REGION Network 7: RD 32002
   RUNG wire#powerrail
      { S7_Templates := "SrcType := Int" } EQ_Contact(in1 := "IEC_Counter_0_DB".CV, in2 := 2)
      { S7_Templates := "[card := 0, word_type := UInt, dword_type := UDInt, byte_type := USInt, any_type := Variant]" } "Modbus_Master_DB".Modbus_Master(REQ := wire#w1, MB_ADDR := 1, MODE := 0, DATA_ADDR := 32002, DATA_LEN := 1, DATA_PTR := "Modbus_Send_Receive_1".Reading_Struct."32002", DONE => "Modbus".Done, BUSY => "Modbus".Busy, ERROR => "Modbus".Error, STATUS => "Modbus".Status)
   END_RUNG
   RUNG wire#powerrail
      Contact( "Comm_ok" )
      { S7_Templates := "SrcType := Int" } EQ_Contact(in1 := "IEC_Counter_0_DB".CV, in2 := 2)
      I_Contact( "Modbus_Master_DB".BUSY )
   END_RUNG wire#w1
   // the same network as SCL:
   IF "IEC_Counter_0_DB".CV = 2 THEN
       "Modbus_Master_DB"(REQ := "Comm_ok" AND ("IEC_Counter_0_DB".CV = 2) AND NOT "Modbus_Master_DB".BUSY,   // Modbus_Master
                          MB_ADDR := 1,
                          MODE := 0,
                          DATA_ADDR := 32002,
                          DATA_LEN := 1,
                          DATA_PTR := "Modbus_Send_Receive_1".Reading_Struct."32002",
                          DONE => "Modbus".Done,
                          BUSY => "Modbus".Busy,
                          ERROR => "Modbus".Error,
                          STATUS => "Modbus".Status);
   END_IF;
END_REGION

REGION Network 8: RD 32003
   RUNG wire#powerrail
      { S7_Templates := "SrcType := Int" } EQ_Contact(in1 := "IEC_Counter_0_DB".CV, in2 := 3)
      { S7_Templates := "[card := 0, word_type := UInt, dword_type := UDInt, byte_type := USInt, any_type := Variant]" } "Modbus_Master_DB".Modbus_Master(REQ := wire#w1, MB_ADDR := 1, MODE := 0, DATA_ADDR := 32003, DATA_LEN := 1, DATA_PTR := "Modbus_Send_Receive_1".Reading_Struct."32003", DONE => "Modbus".Done, BUSY => "Modbus".Busy, ERROR => "Modbus".Error, STATUS => "Modbus".Status)
   END_RUNG
   RUNG wire#powerrail
      Contact( "Comm_ok" )
      { S7_Templates := "SrcType := Int" } EQ_Contact(in1 := "IEC_Counter_0_DB".CV, in2 := 3)
      I_Contact( "Modbus_Master_DB".BUSY )
   END_RUNG wire#w1
   // the same network as SCL:
   IF "IEC_Counter_0_DB".CV = 3 THEN
       "Modbus_Master_DB"(REQ := "Comm_ok" AND ("IEC_Counter_0_DB".CV = 3) AND NOT "Modbus_Master_DB".BUSY,   // Modbus_Master
                          MB_ADDR := 1,
                          MODE := 0,
                          DATA_ADDR := 32003,
                          DATA_LEN := 1,
                          DATA_PTR := "Modbus_Send_Receive_1".Reading_Struct."32003",
                          DONE => "Modbus".Done,
                          BUSY => "Modbus".Busy,
                          ERROR => "Modbus".Error,
                          STATUS => "Modbus".Status);
   END_IF;
END_REGION

REGION Network 9: RD 32004
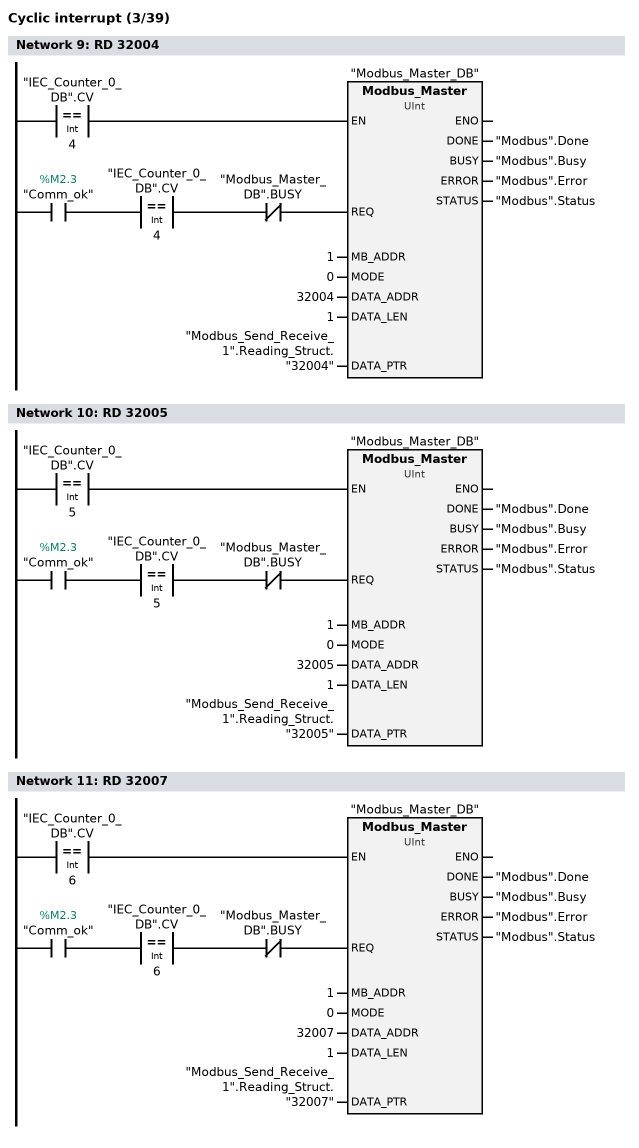
   RUNG wire#powerrail
      { S7_Templates := "SrcType := Int" } EQ_Contact(in1 := "IEC_Counter_0_DB".CV, in2 := 4)
      { S7_Templates := "[card := 0, word_type := UInt, dword_type := UDInt, byte_type := USInt, any_type := Variant]" } "Modbus_Master_DB".Modbus_Master(REQ := wire#w1, MB_ADDR := 1, MODE := 0, DATA_ADDR := 32004, DATA_LEN := 1, DATA_PTR := "Modbus_Send_Receive_1".Reading_Struct."32004", DONE => "Modbus".Done, BUSY => "Modbus".Busy, ERROR => "Modbus".Error, STATUS => "Modbus".Status)
   END_RUNG
   RUNG wire#powerrail
      Contact( "Comm_ok" )
      { S7_Templates := "SrcType := Int" } EQ_Contact(in1 := "IEC_Counter_0_DB".CV, in2 := 4)
      I_Contact( "Modbus_Master_DB".BUSY )
   END_RUNG wire#w1
   // the same network as SCL:
   IF "IEC_Counter_0_DB".CV = 4 THEN
       "Modbus_Master_DB"(REQ := "Comm_ok" AND ("IEC_Counter_0_DB".CV = 4) AND NOT "Modbus_Master_DB".BUSY,   // Modbus_Master
                          MB_ADDR := 1,
                          MODE := 0,
                          DATA_ADDR := 32004,
                          DATA_LEN := 1,
                          DATA_PTR := "Modbus_Send_Receive_1".Reading_Struct."32004",
                          DONE => "Modbus".Done,
                          BUSY => "Modbus".Busy,
                          ERROR => "Modbus".Error,
                          STATUS => "Modbus".Status);
   END_IF;
END_REGION

REGION Network 10: RD 32005
   RUNG wire#powerrail
      { S7_Templates := "SrcType := Int" } EQ_Contact(in1 := "IEC_Counter_0_DB".CV, in2 := 5)
      { S7_Templates := "[card := 0, word_type := UInt, dword_type := UDInt, byte_type := USInt, any_type := Variant]" } "Modbus_Master_DB".Modbus_Master(REQ := wire#w1, MB_ADDR := 1, MODE := 0, DATA_ADDR := 32005, DATA_LEN := 1, DATA_PTR := "Modbus_Send_Receive_1".Reading_Struct."32005", DONE => "Modbus".Done, BUSY => "Modbus".Busy, ERROR => "Modbus".Error, STATUS => "Modbus".Status)
   END_RUNG
   RUNG wire#powerrail
      Contact( "Comm_ok" )
      { S7_Templates := "SrcType := Int" } EQ_Contact(in1 := "IEC_Counter_0_DB".CV, in2 := 5)
      I_Contact( "Modbus_Master_DB".BUSY )
   END_RUNG wire#w1
   // the same network as SCL:
   IF "IEC_Counter_0_DB".CV = 5 THEN
       "Modbus_Master_DB"(REQ := "Comm_ok" AND ("IEC_Counter_0_DB".CV = 5) AND NOT "Modbus_Master_DB".BUSY,   // Modbus_Master
                          MB_ADDR := 1,
                          MODE := 0,
                          DATA_ADDR := 32005,
                          DATA_LEN := 1,
                          DATA_PTR := "Modbus_Send_Receive_1".Reading_Struct."32005",
                          DONE => "Modbus".Done,
                          BUSY => "Modbus".Busy,
                          ERROR => "Modbus".Error,
                          STATUS => "Modbus".Status);
   END_IF;
END_REGION

REGION Network 11: RD 32007
   RUNG wire#powerrail
      { S7_Templates := "SrcType := Int" } EQ_Contact(in1 := "IEC_Counter_0_DB".CV, in2 := 6)
      { S7_Templates := "[card := 0, word_type := UInt, dword_type := UDInt, byte_type := USInt, any_type := Variant]" } "Modbus_Master_DB".Modbus_Master(REQ := wire#w1, MB_ADDR := 1, MODE := 0, DATA_ADDR := 32007, DATA_LEN := 1, DATA_PTR := "Modbus_Send_Receive_1".Reading_Struct."32007", DONE => "Modbus".Done, BUSY => "Modbus".Busy, ERROR => "Modbus".Error, STATUS => "Modbus".Status)
   END_RUNG
   RUNG wire#powerrail
      Contact( "Comm_ok" )
      { S7_Templates := "SrcType := Int" } EQ_Contact(in1 := "IEC_Counter_0_DB".CV, in2 := 6)
      I_Contact( "Modbus_Master_DB".BUSY )
   END_RUNG wire#w1
   // the same network as SCL:
   IF "IEC_Counter_0_DB".CV = 6 THEN
       "Modbus_Master_DB"(REQ := "Comm_ok" AND ("IEC_Counter_0_DB".CV = 6) AND NOT "Modbus_Master_DB".BUSY,   // Modbus_Master
                          MB_ADDR := 1,
                          MODE := 0,
                          DATA_ADDR := 32007,
                          DATA_LEN := 1,
                          DATA_PTR := "Modbus_Send_Receive_1".Reading_Struct."32007",
                          DONE => "Modbus".Done,
                          BUSY => "Modbus".Busy,
                          ERROR => "Modbus".Error,
                          STATUS => "Modbus".Status);
   END_IF;
END_REGION

REGION Network 12: RD 32008
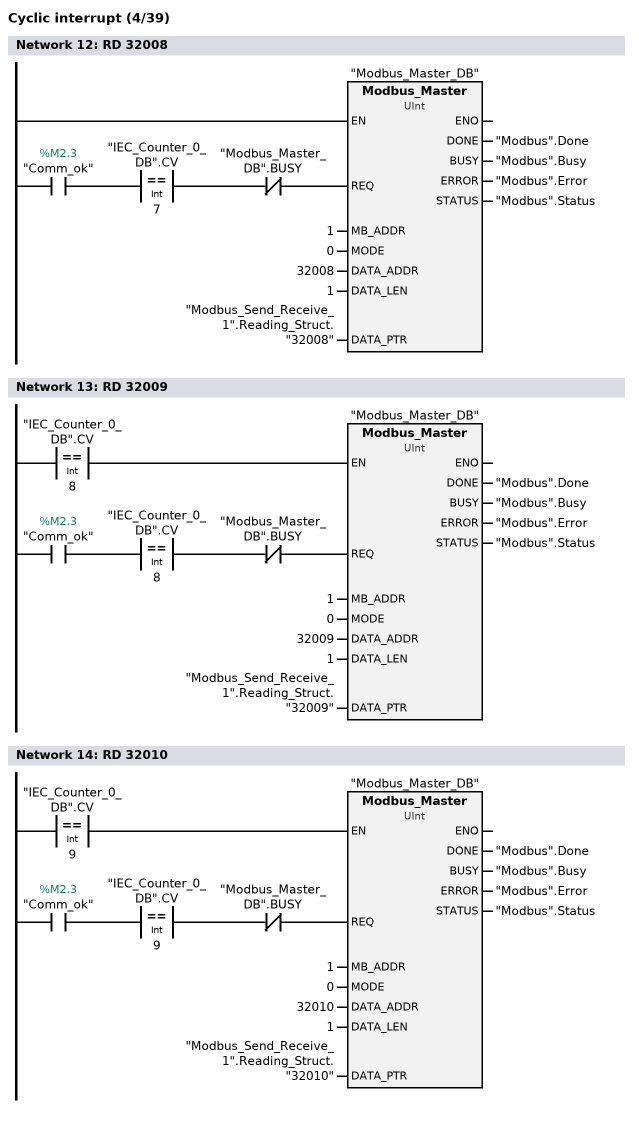
   RUNG wire#powerrail
      { S7_Templates := "[card := 0, word_type := UInt, dword_type := UDInt, byte_type := USInt, any_type := Variant]" } "Modbus_Master_DB".Modbus_Master(REQ := wire#w1, MB_ADDR := 1, MODE := 0, DATA_ADDR := 32008, DATA_LEN := 1, DATA_PTR := "Modbus_Send_Receive_1".Reading_Struct."32008", DONE => "Modbus".Done, BUSY => "Modbus".Busy, ERROR => "Modbus".Error, STATUS => "Modbus".Status)
   END_RUNG
   RUNG wire#powerrail
      Contact( "Comm_ok" )
      { S7_Templates := "SrcType := Int" } EQ_Contact(in1 := "IEC_Counter_0_DB".CV, in2 := 7)
      I_Contact( "Modbus_Master_DB".BUSY )
   END_RUNG wire#w1
   // the same network as SCL:
   "Modbus_Master_DB"(REQ := "Comm_ok" AND ("IEC_Counter_0_DB".CV = 7) AND NOT "Modbus_Master_DB".BUSY,   // Modbus_Master
                      MB_ADDR := 1,
                      MODE := 0,
                      DATA_ADDR := 32008,
                      DATA_LEN := 1,
                      DATA_PTR := "Modbus_Send_Receive_1".Reading_Struct."32008",
                      DONE => "Modbus".Done,
                      BUSY => "Modbus".Busy,
                      ERROR => "Modbus".Error,
                      STATUS => "Modbus".Status);
END_REGION

REGION Network 13: RD 32009
   RUNG wire#powerrail
      { S7_Templates := "SrcType := Int" } EQ_Contact(in1 := "IEC_Counter_0_DB".CV, in2 := 8)
      { S7_Templates := "[card := 0, word_type := UInt, dword_type := UDInt, byte_type := USInt, any_type := Variant]" } "Modbus_Master_DB".Modbus_Master(REQ := wire#w1, MB_ADDR := 1, MODE := 0, DATA_ADDR := 32009, DATA_LEN := 1, DATA_PTR := "Modbus_Send_Receive_1".Reading_Struct."32009", DONE => "Modbus".Done, BUSY => "Modbus".Busy, ERROR => "Modbus".Error, STATUS => "Modbus".Status)
   END_RUNG
   RUNG wire#powerrail
      Contact( "Comm_ok" )
      { S7_Templates := "SrcType := Int" } EQ_Contact(in1 := "IEC_Counter_0_DB".CV, in2 := 8)
      I_Contact( "Modbus_Master_DB".BUSY )
   END_RUNG wire#w1
   // the same network as SCL:
   IF "IEC_Counter_0_DB".CV = 8 THEN
       "Modbus_Master_DB"(REQ := "Comm_ok" AND ("IEC_Counter_0_DB".CV = 8) AND NOT "Modbus_Master_DB".BUSY,   // Modbus_Master
                          MB_ADDR := 1,
                          MODE := 0,
                          DATA_ADDR := 32009,
                          DATA_LEN := 1,
                          DATA_PTR := "Modbus_Send_Receive_1".Reading_Struct."32009",
                          DONE => "Modbus".Done,
                          BUSY => "Modbus".Busy,
                          ERROR => "Modbus".Error,
                          STATUS => "Modbus".Status);
   END_IF;
END_REGION

REGION Network 14: RD 32010
   RUNG wire#powerrail
      { S7_Templates := "SrcType := Int" } EQ_Contact(in1 := "IEC_Counter_0_DB".CV, in2 := 9)
      { S7_Templates := "[card := 0, word_type := UInt, dword_type := UDInt, byte_type := USInt, any_type := Variant]" } "Modbus_Master_DB".Modbus_Master(REQ := wire#w1, MB_ADDR := 1, MODE := 0, DATA_ADDR := 32010, DATA_LEN := 1, DATA_PTR := "Modbus_Send_Receive_1".Reading_Struct."32010", DONE => "Modbus".Done, BUSY => "Modbus".Busy, ERROR => "Modbus".Error, STATUS => "Modbus".Status)
   END_RUNG
   RUNG wire#powerrail
      Contact( "Comm_ok" )
      { S7_Templates := "SrcType := Int" } EQ_Contact(in1 := "IEC_Counter_0_DB".CV, in2 := 9)
      I_Contact( "Modbus_Master_DB".BUSY )
   END_RUNG wire#w1
   // the same network as SCL:
   IF "IEC_Counter_0_DB".CV = 9 THEN
       "Modbus_Master_DB"(REQ := "Comm_ok" AND ("IEC_Counter_0_DB".CV = 9) AND NOT "Modbus_Master_DB".BUSY,   // Modbus_Master
                          MB_ADDR := 1,
                          MODE := 0,
                          DATA_ADDR := 32010,
                          DATA_LEN := 1,
                          DATA_PTR := "Modbus_Send_Receive_1".Reading_Struct."32010",
                          DONE => "Modbus".Done,
                          BUSY => "Modbus".Busy,
                          ERROR => "Modbus".Error,
                          STATUS => "Modbus".Status);
   END_IF;
END_REGION

REGION Network 15: RD 32011
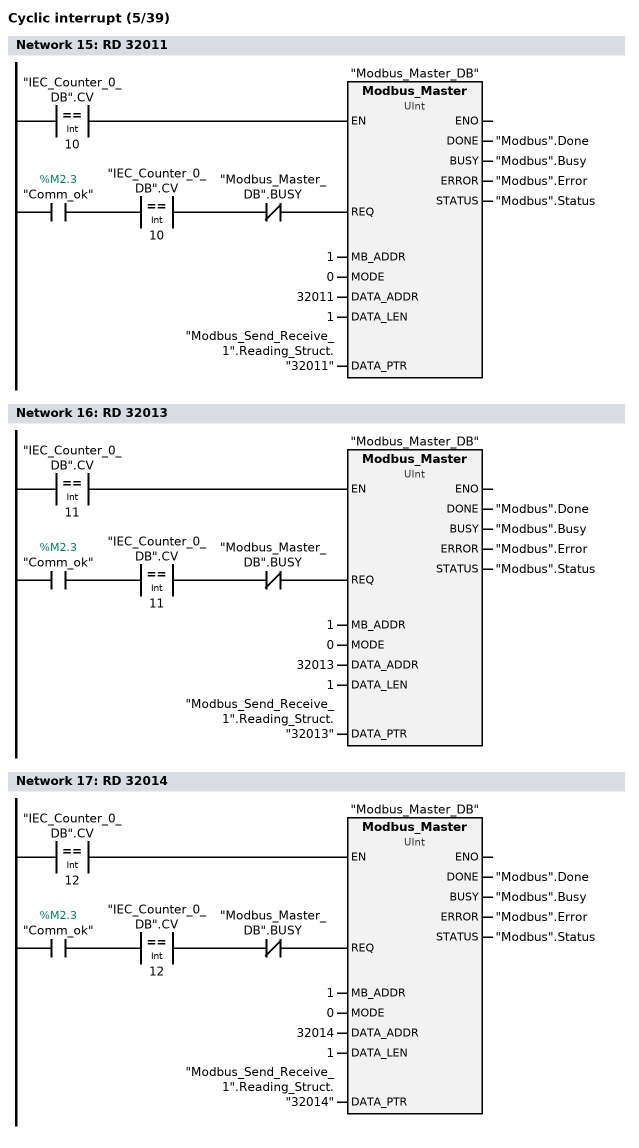
   RUNG wire#powerrail
      { S7_Templates := "SrcType := Int" } EQ_Contact(in1 := "IEC_Counter_0_DB".CV, in2 := 10)
      { S7_Templates := "[card := 0, word_type := UInt, dword_type := UDInt, byte_type := USInt, any_type := Variant]" } "Modbus_Master_DB".Modbus_Master(REQ := wire#w1, MB_ADDR := 1, MODE := 0, DATA_ADDR := 32011, DATA_LEN := 1, DATA_PTR := "Modbus_Send_Receive_1".Reading_Struct."32011", DONE => "Modbus".Done, BUSY => "Modbus".Busy, ERROR => "Modbus".Error, STATUS => "Modbus".Status)
   END_RUNG
   RUNG wire#powerrail
      Contact( "Comm_ok" )
      { S7_Templates := "SrcType := Int" } EQ_Contact(in1 := "IEC_Counter_0_DB".CV, in2 := 10)
      I_Contact( "Modbus_Master_DB".BUSY )
   END_RUNG wire#w1
   // the same network as SCL:
   IF "IEC_Counter_0_DB".CV = 10 THEN
       "Modbus_Master_DB"(REQ := "Comm_ok" AND ("IEC_Counter_0_DB".CV = 10) AND NOT "Modbus_Master_DB".BUSY,   // Modbus_Master
                          MB_ADDR := 1,
                          MODE := 0,
                          DATA_ADDR := 32011,
                          DATA_LEN := 1,
                          DATA_PTR := "Modbus_Send_Receive_1".Reading_Struct."32011",
                          DONE => "Modbus".Done,
                          BUSY => "Modbus".Busy,
                          ERROR => "Modbus".Error,
                          STATUS => "Modbus".Status);
   END_IF;
END_REGION

REGION Network 16: RD 32013
   RUNG wire#powerrail
      { S7_Templates := "SrcType := Int" } EQ_Contact(in1 := "IEC_Counter_0_DB".CV, in2 := 11)
      { S7_Templates := "[card := 0, word_type := UInt, dword_type := UDInt, byte_type := USInt, any_type := Variant]" } "Modbus_Master_DB".Modbus_Master(REQ := wire#w1, MB_ADDR := 1, MODE := 0, DATA_ADDR := 32013, DATA_LEN := 1, DATA_PTR := "Modbus_Send_Receive_1".Reading_Struct."32013", DONE => "Modbus".Done, BUSY => "Modbus".Busy, ERROR => "Modbus".Error, STATUS => "Modbus".Status)
   END_RUNG
   RUNG wire#powerrail
      Contact( "Comm_ok" )
      { S7_Templates := "SrcType := Int" } EQ_Contact(in1 := "IEC_Counter_0_DB".CV, in2 := 11)
      I_Contact( "Modbus_Master_DB".BUSY )
   END_RUNG wire#w1
   // the same network as SCL:
   IF "IEC_Counter_0_DB".CV = 11 THEN
       "Modbus_Master_DB"(REQ := "Comm_ok" AND ("IEC_Counter_0_DB".CV = 11) AND NOT "Modbus_Master_DB".BUSY,   // Modbus_Master
                          MB_ADDR := 1,
                          MODE := 0,
                          DATA_ADDR := 32013,
                          DATA_LEN := 1,
                          DATA_PTR := "Modbus_Send_Receive_1".Reading_Struct."32013",
                          DONE => "Modbus".Done,
                          BUSY => "Modbus".Busy,
                          ERROR => "Modbus".Error,
                          STATUS => "Modbus".Status);
   END_IF;
END_REGION

REGION Network 17: RD 32014
   RUNG wire#powerrail
      { S7_Templates := "SrcType := Int" } EQ_Contact(in1 := "IEC_Counter_0_DB".CV, in2 := 12)
      { S7_Templates := "[card := 0, word_type := UInt, dword_type := UDInt, byte_type := USInt, any_type := Variant]" } "Modbus_Master_DB".Modbus_Master(REQ := wire#w1, MB_ADDR := 1, MODE := 0, DATA_ADDR := 32014, DATA_LEN := 1, DATA_PTR := "Modbus_Send_Receive_1".Reading_Struct."32014", DONE => "Modbus".Done, BUSY => "Modbus".Busy, ERROR => "Modbus".Error, STATUS => "Modbus".Status)
   END_RUNG
   RUNG wire#powerrail
      Contact( "Comm_ok" )
      { S7_Templates := "SrcType := Int" } EQ_Contact(in1 := "IEC_Counter_0_DB".CV, in2 := 12)
      I_Contact( "Modbus_Master_DB".BUSY )
   END_RUNG wire#w1
   // the same network as SCL:
   IF "IEC_Counter_0_DB".CV = 12 THEN
       "Modbus_Master_DB"(REQ := "Comm_ok" AND ("IEC_Counter_0_DB".CV = 12) AND NOT "Modbus_Master_DB".BUSY,   // Modbus_Master
                          MB_ADDR := 1,
                          MODE := 0,
                          DATA_ADDR := 32014,
                          DATA_LEN := 1,
                          DATA_PTR := "Modbus_Send_Receive_1".Reading_Struct."32014",
                          DONE => "Modbus".Done,
                          BUSY => "Modbus".Busy,
                          ERROR => "Modbus".Error,
                          STATUS => "Modbus".Status);
   END_IF;
END_REGION

REGION Network 18: RD 32015
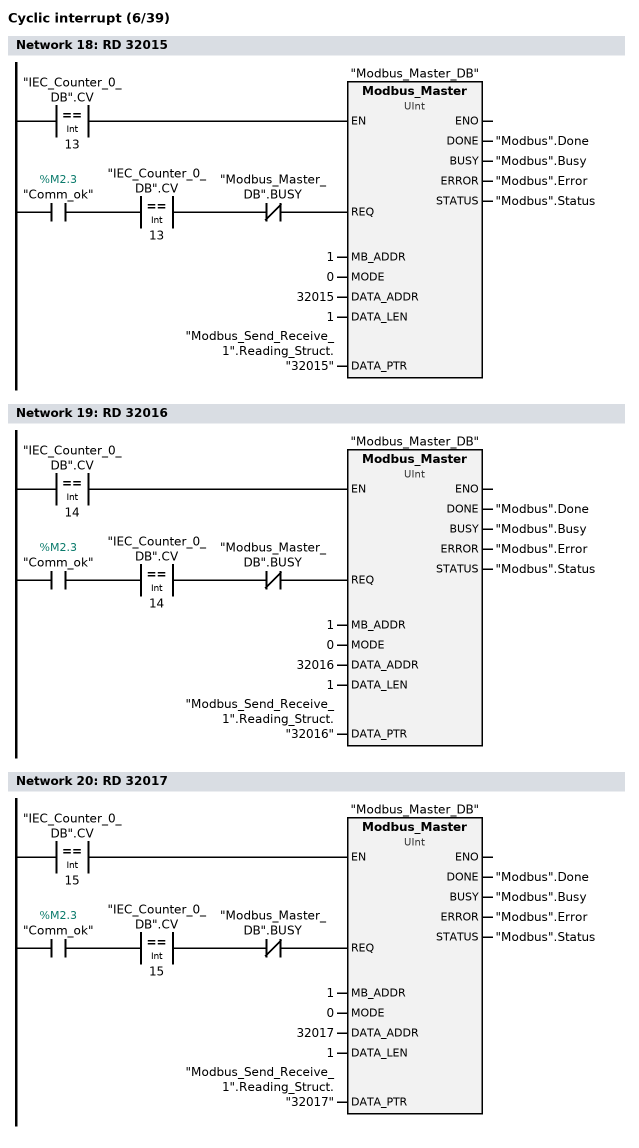
   RUNG wire#powerrail
      { S7_Templates := "SrcType := Int" } EQ_Contact(in1 := "IEC_Counter_0_DB".CV, in2 := 13)
      { S7_Templates := "[card := 0, word_type := UInt, dword_type := UDInt, byte_type := USInt, any_type := Variant]" } "Modbus_Master_DB".Modbus_Master(REQ := wire#w1, MB_ADDR := 1, MODE := 0, DATA_ADDR := 32015, DATA_LEN := 1, DATA_PTR := "Modbus_Send_Receive_1".Reading_Struct."32015", DONE => "Modbus".Done, BUSY => "Modbus".Busy, ERROR => "Modbus".Error, STATUS => "Modbus".Status)
   END_RUNG
   RUNG wire#powerrail
      Contact( "Comm_ok" )
      { S7_Templates := "SrcType := Int" } EQ_Contact(in1 := "IEC_Counter_0_DB".CV, in2 := 13)
      I_Contact( "Modbus_Master_DB".BUSY )
   END_RUNG wire#w1
   // the same network as SCL:
   IF "IEC_Counter_0_DB".CV = 13 THEN
       "Modbus_Master_DB"(REQ := "Comm_ok" AND ("IEC_Counter_0_DB".CV = 13) AND NOT "Modbus_Master_DB".BUSY,   // Modbus_Master
                          MB_ADDR := 1,
                          MODE := 0,
                          DATA_ADDR := 32015,
                          DATA_LEN := 1,
                          DATA_PTR := "Modbus_Send_Receive_1".Reading_Struct."32015",
                          DONE => "Modbus".Done,
                          BUSY => "Modbus".Busy,
                          ERROR => "Modbus".Error,
                          STATUS => "Modbus".Status);
   END_IF;
END_REGION

REGION Network 19: RD 32016
   RUNG wire#powerrail
      { S7_Templates := "SrcType := Int" } EQ_Contact(in1 := "IEC_Counter_0_DB".CV, in2 := 14)
      { S7_Templates := "[card := 0, word_type := UInt, dword_type := UDInt, byte_type := USInt, any_type := Variant]" } "Modbus_Master_DB".Modbus_Master(REQ := wire#w1, MB_ADDR := 1, MODE := 0, DATA_ADDR := 32016, DATA_LEN := 1, DATA_PTR := "Modbus_Send_Receive_1".Reading_Struct."32016", DONE => "Modbus".Done, BUSY => "Modbus".Busy, ERROR => "Modbus".Error, STATUS => "Modbus".Status)
   END_RUNG
   RUNG wire#powerrail
      Contact( "Comm_ok" )
      { S7_Templates := "SrcType := Int" } EQ_Contact(in1 := "IEC_Counter_0_DB".CV, in2 := 14)
      I_Contact( "Modbus_Master_DB".BUSY )
   END_RUNG wire#w1
   // the same network as SCL:
   IF "IEC_Counter_0_DB".CV = 14 THEN
       "Modbus_Master_DB"(REQ := "Comm_ok" AND ("IEC_Counter_0_DB".CV = 14) AND NOT "Modbus_Master_DB".BUSY,   // Modbus_Master
                          MB_ADDR := 1,
                          MODE := 0,
                          DATA_ADDR := 32016,
                          DATA_LEN := 1,
                          DATA_PTR := "Modbus_Send_Receive_1".Reading_Struct."32016",
                          DONE => "Modbus".Done,
                          BUSY => "Modbus".Busy,
                          ERROR => "Modbus".Error,
                          STATUS => "Modbus".Status);
   END_IF;
END_REGION

REGION Network 20: RD 32017
   RUNG wire#powerrail
      { S7_Templates := "SrcType := Int" } EQ_Contact(in1 := "IEC_Counter_0_DB".CV, in2 := 15)
      { S7_Templates := "[card := 0, word_type := UInt, dword_type := UDInt, byte_type := USInt, any_type := Variant]" } "Modbus_Master_DB".Modbus_Master(REQ := wire#w1, MB_ADDR := 1, MODE := 0, DATA_ADDR := 32017, DATA_LEN := 1, DATA_PTR := "Modbus_Send_Receive_1".Reading_Struct."32017", DONE => "Modbus".Done, BUSY => "Modbus".Busy, ERROR => "Modbus".Error, STATUS => "Modbus".Status)
   END_RUNG
   RUNG wire#powerrail
      Contact( "Comm_ok" )
      { S7_Templates := "SrcType := Int" } EQ_Contact(in1 := "IEC_Counter_0_DB".CV, in2 := 15)
      I_Contact( "Modbus_Master_DB".BUSY )
   END_RUNG wire#w1
   // the same network as SCL:
   IF "IEC_Counter_0_DB".CV = 15 THEN
       "Modbus_Master_DB"(REQ := "Comm_ok" AND ("IEC_Counter_0_DB".CV = 15) AND NOT "Modbus_Master_DB".BUSY,   // Modbus_Master
                          MB_ADDR := 1,
                          MODE := 0,
                          DATA_ADDR := 32017,
                          DATA_LEN := 1,
                          DATA_PTR := "Modbus_Send_Receive_1".Reading_Struct."32017",
                          DONE => "Modbus".Done,
                          BUSY => "Modbus".Busy,
                          ERROR => "Modbus".Error,
                          STATUS => "Modbus".Status);
   END_IF;
END_REGION

REGION Network 21: RD 32019
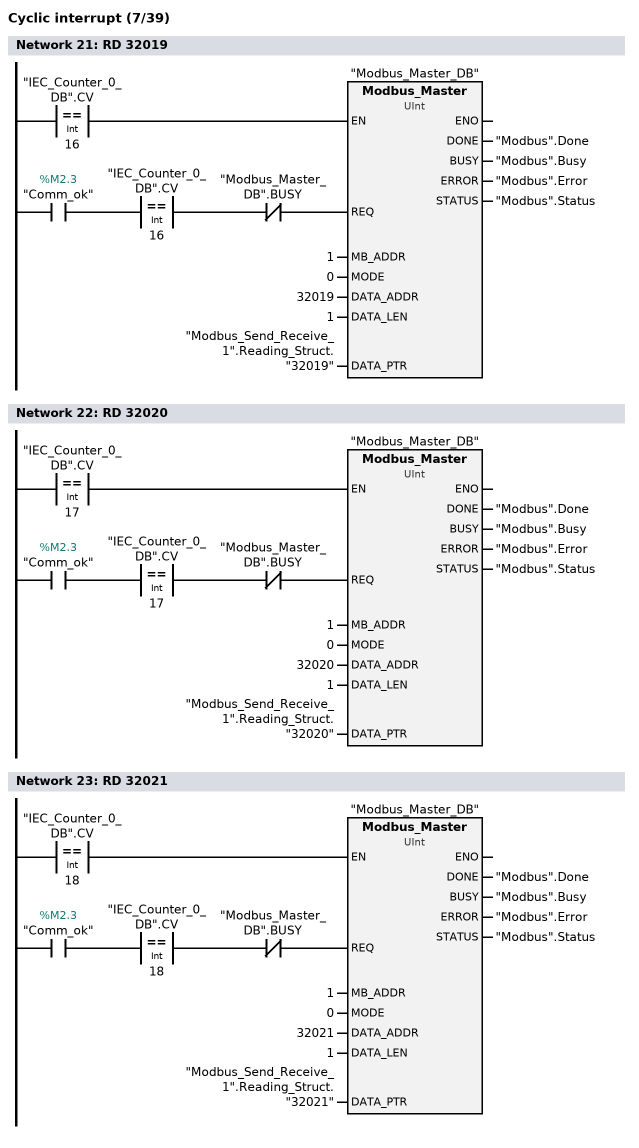
   RUNG wire#powerrail
      { S7_Templates := "SrcType := Int" } EQ_Contact(in1 := "IEC_Counter_0_DB".CV, in2 := 16)
      { S7_Templates := "[card := 0, word_type := UInt, dword_type := UDInt, byte_type := USInt, any_type := Variant]" } "Modbus_Master_DB".Modbus_Master(REQ := wire#w1, MB_ADDR := 1, MODE := 0, DATA_ADDR := 32019, DATA_LEN := 1, DATA_PTR := "Modbus_Send_Receive_1".Reading_Struct."32019", DONE => "Modbus".Done, BUSY => "Modbus".Busy, ERROR => "Modbus".Error, STATUS => "Modbus".Status)
   END_RUNG
   RUNG wire#powerrail
      Contact( "Comm_ok" )
      { S7_Templates := "SrcType := Int" } EQ_Contact(in1 := "IEC_Counter_0_DB".CV, in2 := 16)
      I_Contact( "Modbus_Master_DB".BUSY )
   END_RUNG wire#w1
   // the same network as SCL:
   IF "IEC_Counter_0_DB".CV = 16 THEN
       "Modbus_Master_DB"(REQ := "Comm_ok" AND ("IEC_Counter_0_DB".CV = 16) AND NOT "Modbus_Master_DB".BUSY,   // Modbus_Master
                          MB_ADDR := 1,
                          MODE := 0,
                          DATA_ADDR := 32019,
                          DATA_LEN := 1,
                          DATA_PTR := "Modbus_Send_Receive_1".Reading_Struct."32019",
                          DONE => "Modbus".Done,
                          BUSY => "Modbus".Busy,
                          ERROR => "Modbus".Error,
                          STATUS => "Modbus".Status);
   END_IF;
END_REGION

REGION Network 22: RD 32020
   RUNG wire#powerrail
      { S7_Templates := "SrcType := Int" } EQ_Contact(in1 := "IEC_Counter_0_DB".CV, in2 := 17)
      { S7_Templates := "[card := 0, word_type := UInt, dword_type := UDInt, byte_type := USInt, any_type := Variant]" } "Modbus_Master_DB".Modbus_Master(REQ := wire#w1, MB_ADDR := 1, MODE := 0, DATA_ADDR := 32020, DATA_LEN := 1, DATA_PTR := "Modbus_Send_Receive_1".Reading_Struct."32020", DONE => "Modbus".Done, BUSY => "Modbus".Busy, ERROR => "Modbus".Error, STATUS => "Modbus".Status)
   END_RUNG
   RUNG wire#powerrail
      Contact( "Comm_ok" )
      { S7_Templates := "SrcType := Int" } EQ_Contact(in1 := "IEC_Counter_0_DB".CV, in2 := 17)
      I_Contact( "Modbus_Master_DB".BUSY )
   END_RUNG wire#w1
   // the same network as SCL:
   IF "IEC_Counter_0_DB".CV = 17 THEN
       "Modbus_Master_DB"(REQ := "Comm_ok" AND ("IEC_Counter_0_DB".CV = 17) AND NOT "Modbus_Master_DB".BUSY,   // Modbus_Master
                          MB_ADDR := 1,
                          MODE := 0,
                          DATA_ADDR := 32020,
                          DATA_LEN := 1,
                          DATA_PTR := "Modbus_Send_Receive_1".Reading_Struct."32020",
                          DONE => "Modbus".Done,
                          BUSY => "Modbus".Busy,
                          ERROR => "Modbus".Error,
                          STATUS => "Modbus".Status);
   END_IF;
END_REGION

REGION Network 23: RD 32021
   RUNG wire#powerrail
      { S7_Templates := "SrcType := Int" } EQ_Contact(in1 := "IEC_Counter_0_DB".CV, in2 := 18)
      { S7_Templates := "[card := 0, word_type := UInt, dword_type := UDInt, byte_type := USInt, any_type := Variant]" } "Modbus_Master_DB".Modbus_Master(REQ := wire#w1, MB_ADDR := 1, MODE := 0, DATA_ADDR := 32021, DATA_LEN := 1, DATA_PTR := "Modbus_Send_Receive_1".Reading_Struct."32021", DONE => "Modbus".Done, BUSY => "Modbus".Busy, ERROR => "Modbus".Error, STATUS => "Modbus".Status)
   END_RUNG
   RUNG wire#powerrail
      Contact( "Comm_ok" )
      { S7_Templates := "SrcType := Int" } EQ_Contact(in1 := "IEC_Counter_0_DB".CV, in2 := 18)
      I_Contact( "Modbus_Master_DB".BUSY )
   END_RUNG wire#w1
   // the same network as SCL:
   IF "IEC_Counter_0_DB".CV = 18 THEN
       "Modbus_Master_DB"(REQ := "Comm_ok" AND ("IEC_Counter_0_DB".CV = 18) AND NOT "Modbus_Master_DB".BUSY,   // Modbus_Master
                          MB_ADDR := 1,
                          MODE := 0,
                          DATA_ADDR := 32021,
                          DATA_LEN := 1,
                          DATA_PTR := "Modbus_Send_Receive_1".Reading_Struct."32021",
                          DONE => "Modbus".Done,
                          BUSY => "Modbus".Busy,
                          ERROR => "Modbus".Error,
                          STATUS => "Modbus".Status);
   END_IF;
END_REGION

REGION Network 24: RD 32022
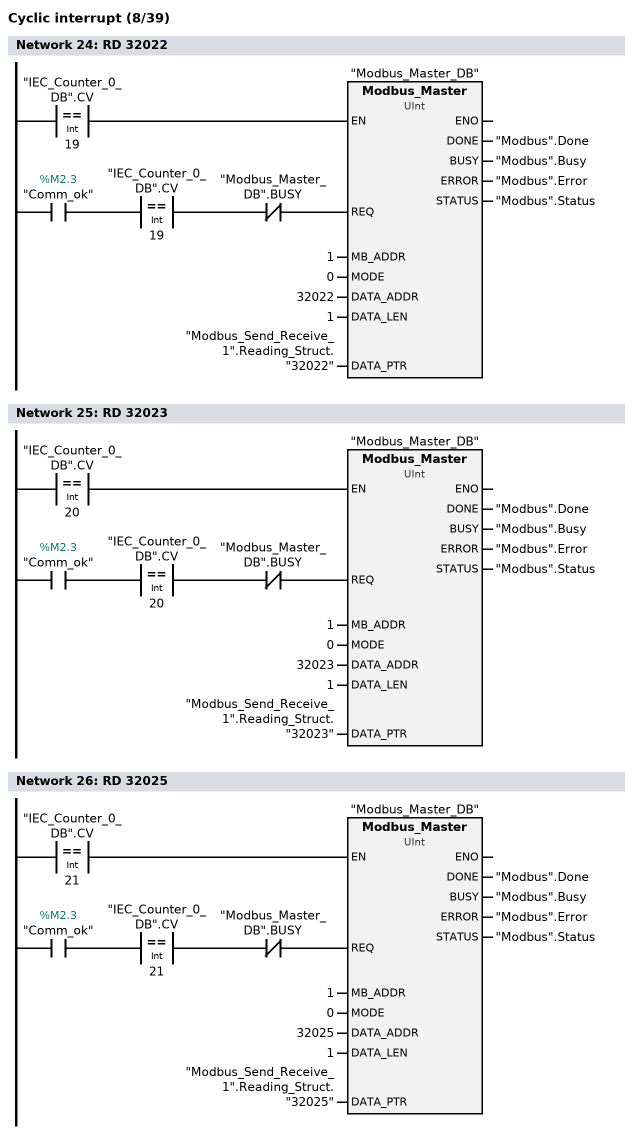
   RUNG wire#powerrail
      { S7_Templates := "SrcType := Int" } EQ_Contact(in1 := "IEC_Counter_0_DB".CV, in2 := 19)
      { S7_Templates := "[card := 0, word_type := UInt, dword_type := UDInt, byte_type := USInt, any_type := Variant]" } "Modbus_Master_DB".Modbus_Master(REQ := wire#w1, MB_ADDR := 1, MODE := 0, DATA_ADDR := 32022, DATA_LEN := 1, DATA_PTR := "Modbus_Send_Receive_1".Reading_Struct."32022", DONE => "Modbus".Done, BUSY => "Modbus".Busy, ERROR => "Modbus".Error, STATUS => "Modbus".Status)
   END_RUNG
   RUNG wire#powerrail
      Contact( "Comm_ok" )
      { S7_Templates := "SrcType := Int" } EQ_Contact(in1 := "IEC_Counter_0_DB".CV, in2 := 19)
      I_Contact( "Modbus_Master_DB".BUSY )
   END_RUNG wire#w1
   // the same network as SCL:
   IF "IEC_Counter_0_DB".CV = 19 THEN
       "Modbus_Master_DB"(REQ := "Comm_ok" AND ("IEC_Counter_0_DB".CV = 19) AND NOT "Modbus_Master_DB".BUSY,   // Modbus_Master
                          MB_ADDR := 1,
                          MODE := 0,
                          DATA_ADDR := 32022,
                          DATA_LEN := 1,
                          DATA_PTR := "Modbus_Send_Receive_1".Reading_Struct."32022",
                          DONE => "Modbus".Done,
                          BUSY => "Modbus".Busy,
                          ERROR => "Modbus".Error,
                          STATUS => "Modbus".Status);
   END_IF;
END_REGION

REGION Network 25: RD 32023
   RUNG wire#powerrail
      { S7_Templates := "SrcType := Int" } EQ_Contact(in1 := "IEC_Counter_0_DB".CV, in2 := 20)
      { S7_Templates := "[card := 0, word_type := UInt, dword_type := UDInt, byte_type := USInt, any_type := Variant]" } "Modbus_Master_DB".Modbus_Master(REQ := wire#w1, MB_ADDR := 1, MODE := 0, DATA_ADDR := 32023, DATA_LEN := 1, DATA_PTR := "Modbus_Send_Receive_1".Reading_Struct."32023", DONE => "Modbus".Done, BUSY => "Modbus".Busy, ERROR => "Modbus".Error, STATUS => "Modbus".Status)
   END_RUNG
   RUNG wire#powerrail
      Contact( "Comm_ok" )
      { S7_Templates := "SrcType := Int" } EQ_Contact(in1 := "IEC_Counter_0_DB".CV, in2 := 20)
      I_Contact( "Modbus_Master_DB".BUSY )
   END_RUNG wire#w1
   // the same network as SCL:
   IF "IEC_Counter_0_DB".CV = 20 THEN
       "Modbus_Master_DB"(REQ := "Comm_ok" AND ("IEC_Counter_0_DB".CV = 20) AND NOT "Modbus_Master_DB".BUSY,   // Modbus_Master
                          MB_ADDR := 1,
                          MODE := 0,
                          DATA_ADDR := 32023,
                          DATA_LEN := 1,
                          DATA_PTR := "Modbus_Send_Receive_1".Reading_Struct."32023",
                          DONE => "Modbus".Done,
                          BUSY => "Modbus".Busy,
                          ERROR => "Modbus".Error,
                          STATUS => "Modbus".Status);
   END_IF;
END_REGION

REGION Network 26: RD 32025
   RUNG wire#powerrail
      { S7_Templates := "SrcType := Int" } EQ_Contact(in1 := "IEC_Counter_0_DB".CV, in2 := 21)
      { S7_Templates := "[card := 0, word_type := UInt, dword_type := UDInt, byte_type := USInt, any_type := Variant]" } "Modbus_Master_DB".Modbus_Master(REQ := wire#w1, MB_ADDR := 1, MODE := 0, DATA_ADDR := 32025, DATA_LEN := 1, DATA_PTR := "Modbus_Send_Receive_1".Reading_Struct."32025", DONE => "Modbus".Done, BUSY => "Modbus".Busy, ERROR => "Modbus".Error, STATUS => "Modbus".Status)
   END_RUNG
   RUNG wire#powerrail
      Contact( "Comm_ok" )
      { S7_Templates := "SrcType := Int" } EQ_Contact(in1 := "IEC_Counter_0_DB".CV, in2 := 21)
      I_Contact( "Modbus_Master_DB".BUSY )
   END_RUNG wire#w1
   // the same network as SCL:
   IF "IEC_Counter_0_DB".CV = 21 THEN
       "Modbus_Master_DB"(REQ := "Comm_ok" AND ("IEC_Counter_0_DB".CV = 21) AND NOT "Modbus_Master_DB".BUSY,   // Modbus_Master
                          MB_ADDR := 1,
                          MODE := 0,
                          DATA_ADDR := 32025,
                          DATA_LEN := 1,
                          DATA_PTR := "Modbus_Send_Receive_1".Reading_Struct."32025",
                          DONE => "Modbus".Done,
                          BUSY => "Modbus".Busy,
                          ERROR => "Modbus".Error,
                          STATUS => "Modbus".Status);
   END_IF;
END_REGION

REGION Network 27: RD 32026
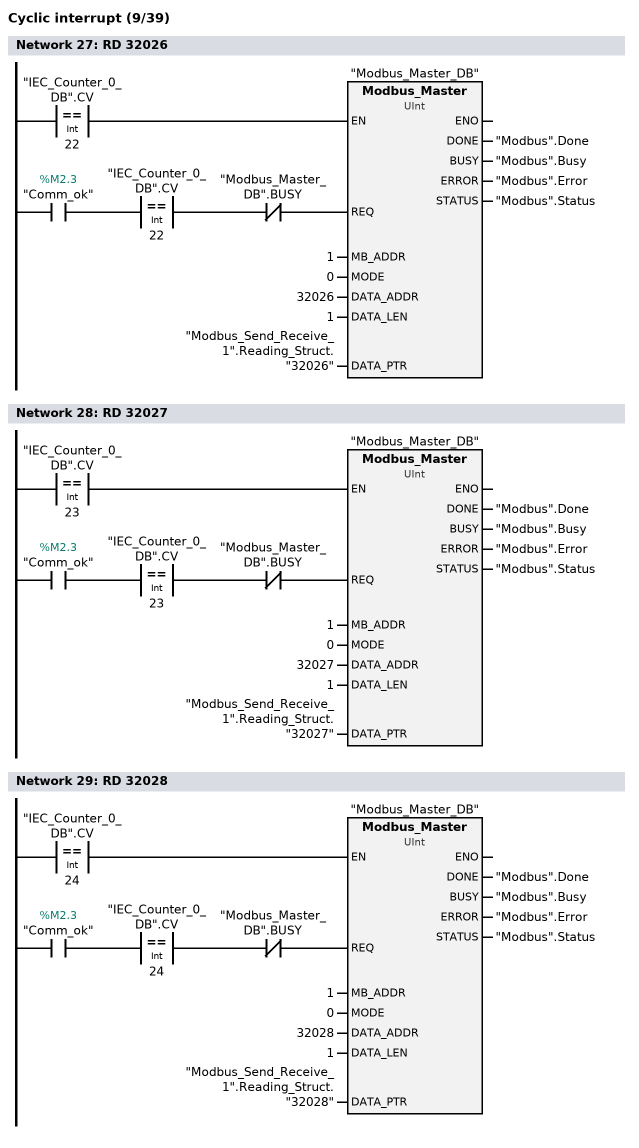
   RUNG wire#powerrail
      { S7_Templates := "SrcType := Int" } EQ_Contact(in1 := "IEC_Counter_0_DB".CV, in2 := 22)
      { S7_Templates := "[card := 0, word_type := UInt, dword_type := UDInt, byte_type := USInt, any_type := Variant]" } "Modbus_Master_DB".Modbus_Master(REQ := wire#w1, MB_ADDR := 1, MODE := 0, DATA_ADDR := 32026, DATA_LEN := 1, DATA_PTR := "Modbus_Send_Receive_1".Reading_Struct."32026", DONE => "Modbus".Done, BUSY => "Modbus".Busy, ERROR => "Modbus".Error, STATUS => "Modbus".Status)
   END_RUNG
   RUNG wire#powerrail
      Contact( "Comm_ok" )
      { S7_Templates := "SrcType := Int" } EQ_Contact(in1 := "IEC_Counter_0_DB".CV, in2 := 22)
      I_Contact( "Modbus_Master_DB".BUSY )
   END_RUNG wire#w1
   // the same network as SCL:
   IF "IEC_Counter_0_DB".CV = 22 THEN
       "Modbus_Master_DB"(REQ := "Comm_ok" AND ("IEC_Counter_0_DB".CV = 22) AND NOT "Modbus_Master_DB".BUSY,   // Modbus_Master
                          MB_ADDR := 1,
                          MODE := 0,
                          DATA_ADDR := 32026,
                          DATA_LEN := 1,
                          DATA_PTR := "Modbus_Send_Receive_1".Reading_Struct."32026",
                          DONE => "Modbus".Done,
                          BUSY => "Modbus".Busy,
                          ERROR => "Modbus".Error,
                          STATUS => "Modbus".Status);
   END_IF;
END_REGION

REGION Network 28: RD 32027
   RUNG wire#powerrail
      { S7_Templates := "SrcType := Int" } EQ_Contact(in1 := "IEC_Counter_0_DB".CV, in2 := 23)
      { S7_Templates := "[card := 0, word_type := UInt, dword_type := UDInt, byte_type := USInt, any_type := Variant]" } "Modbus_Master_DB".Modbus_Master(REQ := wire#w1, MB_ADDR := 1, MODE := 0, DATA_ADDR := 32027, DATA_LEN := 1, DATA_PTR := "Modbus_Send_Receive_1".Reading_Struct."32027", DONE => "Modbus".Done, BUSY => "Modbus".Busy, ERROR => "Modbus".Error, STATUS => "Modbus".Status)
   END_RUNG
   RUNG wire#powerrail
      Contact( "Comm_ok" )
      { S7_Templates := "SrcType := Int" } EQ_Contact(in1 := "IEC_Counter_0_DB".CV, in2 := 23)
      I_Contact( "Modbus_Master_DB".BUSY )
   END_RUNG wire#w1
   // the same network as SCL:
   IF "IEC_Counter_0_DB".CV = 23 THEN
       "Modbus_Master_DB"(REQ := "Comm_ok" AND ("IEC_Counter_0_DB".CV = 23) AND NOT "Modbus_Master_DB".BUSY,   // Modbus_Master
                          MB_ADDR := 1,
                          MODE := 0,
                          DATA_ADDR := 32027,
                          DATA_LEN := 1,
                          DATA_PTR := "Modbus_Send_Receive_1".Reading_Struct."32027",
                          DONE => "Modbus".Done,
                          BUSY => "Modbus".Busy,
                          ERROR => "Modbus".Error,
                          STATUS => "Modbus".Status);
   END_IF;
END_REGION

REGION Network 29: RD 32028
   RUNG wire#powerrail
      { S7_Templates := "SrcType := Int" } EQ_Contact(in1 := "IEC_Counter_0_DB".CV, in2 := 24)
      { S7_Templates := "[card := 0, word_type := UInt, dword_type := UDInt, byte_type := USInt, any_type := Variant]" } "Modbus_Master_DB".Modbus_Master(REQ := wire#w1, MB_ADDR := 1, MODE := 0, DATA_ADDR := 32028, DATA_LEN := 1, DATA_PTR := "Modbus_Send_Receive_1".Reading_Struct."32028", DONE => "Modbus".Done, BUSY => "Modbus".Busy, ERROR => "Modbus".Error, STATUS => "Modbus".Status)
   END_RUNG
   RUNG wire#powerrail
      Contact( "Comm_ok" )
      { S7_Templates := "SrcType := Int" } EQ_Contact(in1 := "IEC_Counter_0_DB".CV, in2 := 24)
      I_Contact( "Modbus_Master_DB".BUSY )
   END_RUNG wire#w1
   // the same network as SCL:
   IF "IEC_Counter_0_DB".CV = 24 THEN
       "Modbus_Master_DB"(REQ := "Comm_ok" AND ("IEC_Counter_0_DB".CV = 24) AND NOT "Modbus_Master_DB".BUSY,   // Modbus_Master
                          MB_ADDR := 1,
                          MODE := 0,
                          DATA_ADDR := 32028,
                          DATA_LEN := 1,
                          DATA_PTR := "Modbus_Send_Receive_1".Reading_Struct."32028",
                          DONE => "Modbus".Done,
                          BUSY => "Modbus".Busy,
                          ERROR => "Modbus".Error,
                          STATUS => "Modbus".Status);
   END_IF;
END_REGION

REGION Network 30: RD 32029
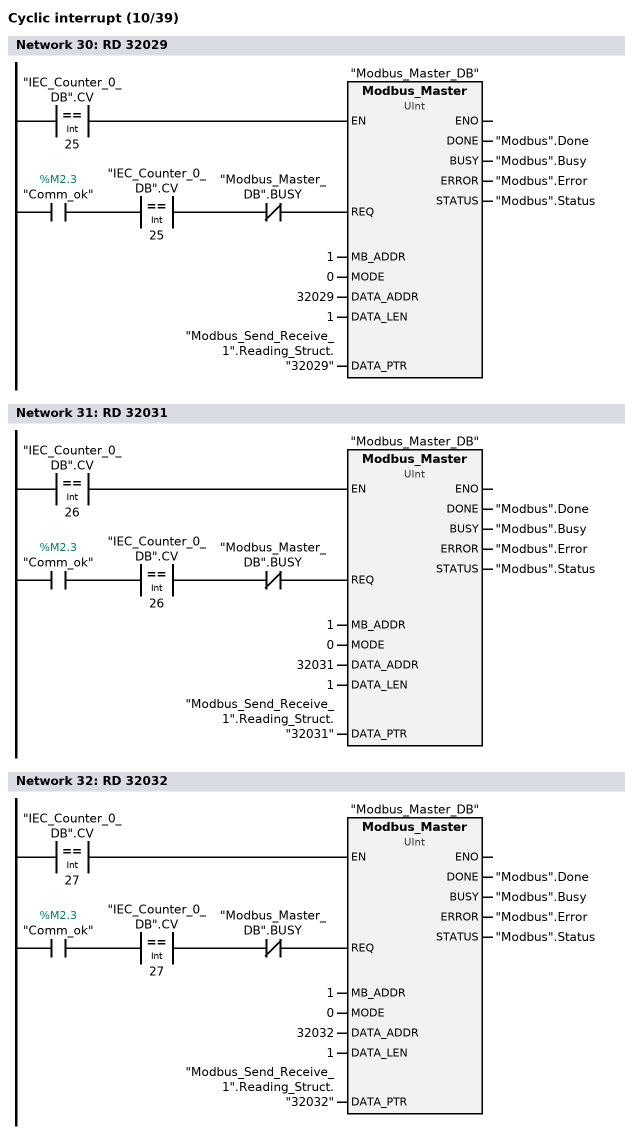
   RUNG wire#powerrail
      { S7_Templates := "SrcType := Int" } EQ_Contact(in1 := "IEC_Counter_0_DB".CV, in2 := 25)
      { S7_Templates := "[card := 0, word_type := UInt, dword_type := UDInt, byte_type := USInt, any_type := Variant]" } "Modbus_Master_DB".Modbus_Master(REQ := wire#w1, MB_ADDR := 1, MODE := 0, DATA_ADDR := 32029, DATA_LEN := 1, DATA_PTR := "Modbus_Send_Receive_1".Reading_Struct."32029", DONE => "Modbus".Done, BUSY => "Modbus".Busy, ERROR => "Modbus".Error, STATUS => "Modbus".Status)
   END_RUNG
   RUNG wire#powerrail
      Contact( "Comm_ok" )
      { S7_Templates := "SrcType := Int" } EQ_Contact(in1 := "IEC_Counter_0_DB".CV, in2 := 25)
      I_Contact( "Modbus_Master_DB".BUSY )
   END_RUNG wire#w1
   // the same network as SCL:
   IF "IEC_Counter_0_DB".CV = 25 THEN
       "Modbus_Master_DB"(REQ := "Comm_ok" AND ("IEC_Counter_0_DB".CV = 25) AND NOT "Modbus_Master_DB".BUSY,   // Modbus_Master
                          MB_ADDR := 1,
                          MODE := 0,
                          DATA_ADDR := 32029,
                          DATA_LEN := 1,
                          DATA_PTR := "Modbus_Send_Receive_1".Reading_Struct."32029",
                          DONE => "Modbus".Done,
                          BUSY => "Modbus".Busy,
                          ERROR => "Modbus".Error,
                          STATUS => "Modbus".Status);
   END_IF;
END_REGION

REGION Network 31: RD 32031
   RUNG wire#powerrail
      { S7_Templates := "SrcType := Int" } EQ_Contact(in1 := "IEC_Counter_0_DB".CV, in2 := 26)
      { S7_Templates := "[card := 0, word_type := UInt, dword_type := UDInt, byte_type := USInt, any_type := Variant]" } "Modbus_Master_DB".Modbus_Master(REQ := wire#w1, MB_ADDR := 1, MODE := 0, DATA_ADDR := 32031, DATA_LEN := 1, DATA_PTR := "Modbus_Send_Receive_1".Reading_Struct."32031", DONE => "Modbus".Done, BUSY => "Modbus".Busy, ERROR => "Modbus".Error, STATUS => "Modbus".Status)
   END_RUNG
   RUNG wire#powerrail
      Contact( "Comm_ok" )
      { S7_Templates := "SrcType := Int" } EQ_Contact(in1 := "IEC_Counter_0_DB".CV, in2 := 26)
      I_Contact( "Modbus_Master_DB".BUSY )
   END_RUNG wire#w1
   // the same network as SCL:
   IF "IEC_Counter_0_DB".CV = 26 THEN
       "Modbus_Master_DB"(REQ := "Comm_ok" AND ("IEC_Counter_0_DB".CV = 26) AND NOT "Modbus_Master_DB".BUSY,   // Modbus_Master
                          MB_ADDR := 1,
                          MODE := 0,
                          DATA_ADDR := 32031,
                          DATA_LEN := 1,
                          DATA_PTR := "Modbus_Send_Receive_1".Reading_Struct."32031",
                          DONE => "Modbus".Done,
                          BUSY => "Modbus".Busy,
                          ERROR => "Modbus".Error,
                          STATUS => "Modbus".Status);
   END_IF;
END_REGION

REGION Network 32: RD 32032
   RUNG wire#powerrail
      { S7_Templates := "SrcType := Int" } EQ_Contact(in1 := "IEC_Counter_0_DB".CV, in2 := 27)
      { S7_Templates := "[card := 0, word_type := UInt, dword_type := UDInt, byte_type := USInt, any_type := Variant]" } "Modbus_Master_DB".Modbus_Master(REQ := wire#w1, MB_ADDR := 1, MODE := 0, DATA_ADDR := 32032, DATA_LEN := 1, DATA_PTR := "Modbus_Send_Receive_1".Reading_Struct."32032", DONE => "Modbus".Done, BUSY => "Modbus".Busy, ERROR => "Modbus".Error, STATUS => "Modbus".Status)
   END_RUNG
   RUNG wire#powerrail
      Contact( "Comm_ok" )
      { S7_Templates := "SrcType := Int" } EQ_Contact(in1 := "IEC_Counter_0_DB".CV, in2 := 27)
      I_Contact( "Modbus_Master_DB".BUSY )
   END_RUNG wire#w1
   // the same network as SCL:
   IF "IEC_Counter_0_DB".CV = 27 THEN
       "Modbus_Master_DB"(REQ := "Comm_ok" AND ("IEC_Counter_0_DB".CV = 27) AND NOT "Modbus_Master_DB".BUSY,   // Modbus_Master
                          MB_ADDR := 1,
                          MODE := 0,
                          DATA_ADDR := 32032,
                          DATA_LEN := 1,
                          DATA_PTR := "Modbus_Send_Receive_1".Reading_Struct."32032",
                          DONE => "Modbus".Done,
                          BUSY => "Modbus".Busy,
                          ERROR => "Modbus".Error,
                          STATUS => "Modbus".Status);
   END_IF;
END_REGION

REGION Network 33: RD 32033
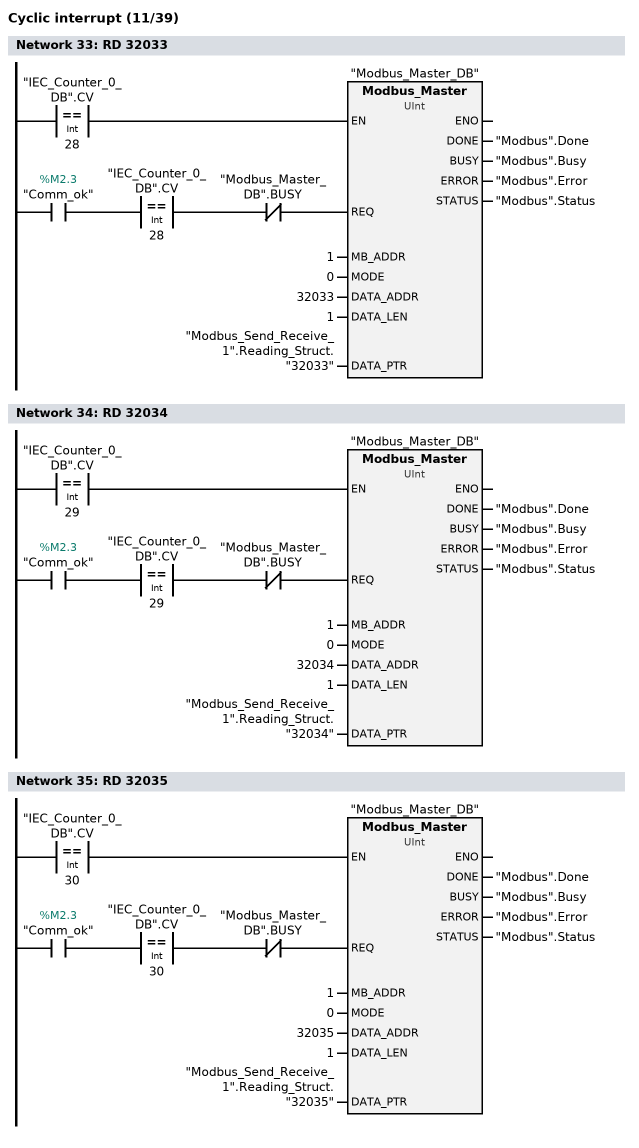
   RUNG wire#powerrail
      { S7_Templates := "SrcType := Int" } EQ_Contact(in1 := "IEC_Counter_0_DB".CV, in2 := 28)
      { S7_Templates := "[card := 0, word_type := UInt, dword_type := UDInt, byte_type := USInt, any_type := Variant]" } "Modbus_Master_DB".Modbus_Master(REQ := wire#w1, MB_ADDR := 1, MODE := 0, DATA_ADDR := 32033, DATA_LEN := 1, DATA_PTR := "Modbus_Send_Receive_1".Reading_Struct."32033", DONE => "Modbus".Done, BUSY => "Modbus".Busy, ERROR => "Modbus".Error, STATUS => "Modbus".Status)
   END_RUNG
   RUNG wire#powerrail
      Contact( "Comm_ok" )
      { S7_Templates := "SrcType := Int" } EQ_Contact(in1 := "IEC_Counter_0_DB".CV, in2 := 28)
      I_Contact( "Modbus_Master_DB".BUSY )
   END_RUNG wire#w1
   // the same network as SCL:
   IF "IEC_Counter_0_DB".CV = 28 THEN
       "Modbus_Master_DB"(REQ := "Comm_ok" AND ("IEC_Counter_0_DB".CV = 28) AND NOT "Modbus_Master_DB".BUSY,   // Modbus_Master
                          MB_ADDR := 1,
                          MODE := 0,
                          DATA_ADDR := 32033,
                          DATA_LEN := 1,
                          DATA_PTR := "Modbus_Send_Receive_1".Reading_Struct."32033",
                          DONE => "Modbus".Done,
                          BUSY => "Modbus".Busy,
                          ERROR => "Modbus".Error,
                          STATUS => "Modbus".Status);
   END_IF;
END_REGION

REGION Network 34: RD 32034
   RUNG wire#powerrail
      { S7_Templates := "SrcType := Int" } EQ_Contact(in1 := "IEC_Counter_0_DB".CV, in2 := 29)
      { S7_Templates := "[card := 0, word_type := UInt, dword_type := UDInt, byte_type := USInt, any_type := Variant]" } "Modbus_Master_DB".Modbus_Master(REQ := wire#w1, MB_ADDR := 1, MODE := 0, DATA_ADDR := 32034, DATA_LEN := 1, DATA_PTR := "Modbus_Send_Receive_1".Reading_Struct."32034", DONE => "Modbus".Done, BUSY => "Modbus".Busy, ERROR => "Modbus".Error, STATUS => "Modbus".Status)
   END_RUNG
   RUNG wire#powerrail
      Contact( "Comm_ok" )
      { S7_Templates := "SrcType := Int" } EQ_Contact(in1 := "IEC_Counter_0_DB".CV, in2 := 29)
      I_Contact( "Modbus_Master_DB".BUSY )
   END_RUNG wire#w1
   // the same network as SCL:
   IF "IEC_Counter_0_DB".CV = 29 THEN
       "Modbus_Master_DB"(REQ := "Comm_ok" AND ("IEC_Counter_0_DB".CV = 29) AND NOT "Modbus_Master_DB".BUSY,   // Modbus_Master
                          MB_ADDR := 1,
                          MODE := 0,
                          DATA_ADDR := 32034,
                          DATA_LEN := 1,
                          DATA_PTR := "Modbus_Send_Receive_1".Reading_Struct."32034",
                          DONE => "Modbus".Done,
                          BUSY => "Modbus".Busy,
                          ERROR => "Modbus".Error,
                          STATUS => "Modbus".Status);
   END_IF;
END_REGION

REGION Network 35: RD 32035
   RUNG wire#powerrail
      { S7_Templates := "SrcType := Int" } EQ_Contact(in1 := "IEC_Counter_0_DB".CV, in2 := 30)
      { S7_Templates := "[card := 0, word_type := UInt, dword_type := UDInt, byte_type := USInt, any_type := Variant]" } "Modbus_Master_DB".Modbus_Master(REQ := wire#w1, MB_ADDR := 1, MODE := 0, DATA_ADDR := 32035, DATA_LEN := 1, DATA_PTR := "Modbus_Send_Receive_1".Reading_Struct."32035", DONE => "Modbus".Done, BUSY => "Modbus".Busy, ERROR => "Modbus".Error, STATUS => "Modbus".Status)
   END_RUNG
   RUNG wire#powerrail
      Contact( "Comm_ok" )
      { S7_Templates := "SrcType := Int" } EQ_Contact(in1 := "IEC_Counter_0_DB".CV, in2 := 30)
      I_Contact( "Modbus_Master_DB".BUSY )
   END_RUNG wire#w1
   // the same network as SCL:
   IF "IEC_Counter_0_DB".CV = 30 THEN
       "Modbus_Master_DB"(REQ := "Comm_ok" AND ("IEC_Counter_0_DB".CV = 30) AND NOT "Modbus_Master_DB".BUSY,   // Modbus_Master
                          MB_ADDR := 1,
                          MODE := 0,
                          DATA_ADDR := 32035,
                          DATA_LEN := 1,
                          DATA_PTR := "Modbus_Send_Receive_1".Reading_Struct."32035",
                          DONE => "Modbus".Done,
                          BUSY => "Modbus".Busy,
                          ERROR => "Modbus".Error,
                          STATUS => "Modbus".Status);
   END_IF;
END_REGION

REGION Network 36: RD 32037
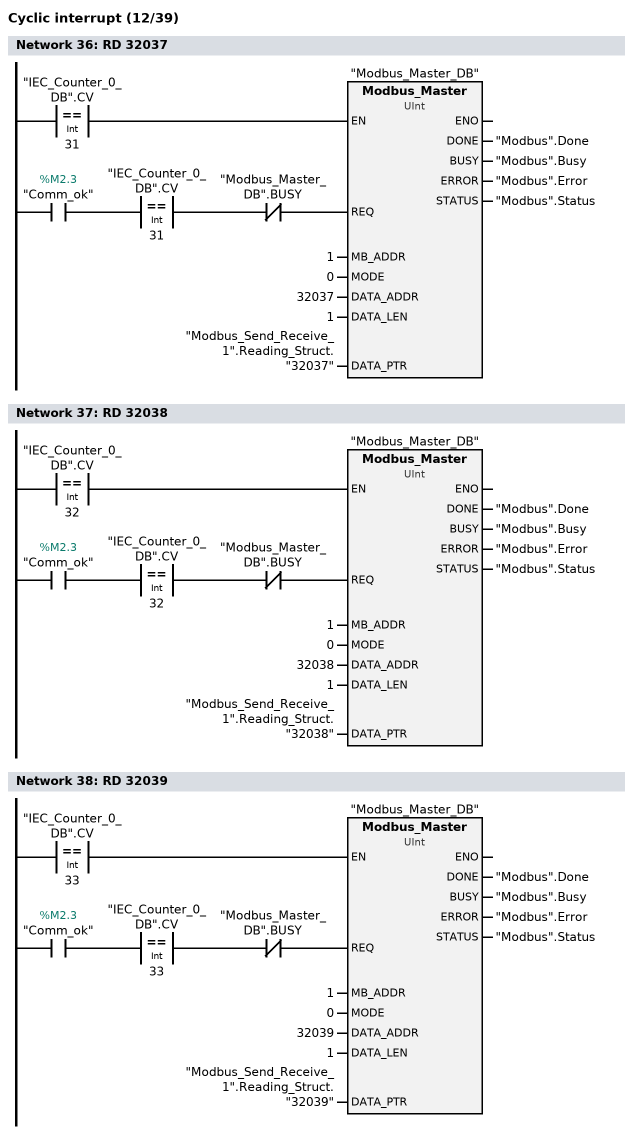
   RUNG wire#powerrail
      { S7_Templates := "SrcType := Int" } EQ_Contact(in1 := "IEC_Counter_0_DB".CV, in2 := 31)
      { S7_Templates := "[card := 0, word_type := UInt, dword_type := UDInt, byte_type := USInt, any_type := Variant]" } "Modbus_Master_DB".Modbus_Master(REQ := wire#w1, MB_ADDR := 1, MODE := 0, DATA_ADDR := 32037, DATA_LEN := 1, DATA_PTR := "Modbus_Send_Receive_1".Reading_Struct."32037", DONE => "Modbus".Done, BUSY => "Modbus".Busy, ERROR => "Modbus".Error, STATUS => "Modbus".Status)
   END_RUNG
   RUNG wire#powerrail
      Contact( "Comm_ok" )
      { S7_Templates := "SrcType := Int" } EQ_Contact(in1 := "IEC_Counter_0_DB".CV, in2 := 31)
      I_Contact( "Modbus_Master_DB".BUSY )
   END_RUNG wire#w1
   // the same network as SCL:
   IF "IEC_Counter_0_DB".CV = 31 THEN
       "Modbus_Master_DB"(REQ := "Comm_ok" AND ("IEC_Counter_0_DB".CV = 31) AND NOT "Modbus_Master_DB".BUSY,   // Modbus_Master
                          MB_ADDR := 1,
                          MODE := 0,
                          DATA_ADDR := 32037,
                          DATA_LEN := 1,
                          DATA_PTR := "Modbus_Send_Receive_1".Reading_Struct."32037",
                          DONE => "Modbus".Done,
                          BUSY => "Modbus".Busy,
                          ERROR => "Modbus".Error,
                          STATUS => "Modbus".Status);
   END_IF;
END_REGION

REGION Network 37: RD 32038
   RUNG wire#powerrail
      { S7_Templates := "SrcType := Int" } EQ_Contact(in1 := "IEC_Counter_0_DB".CV, in2 := 32)
      { S7_Templates := "[card := 0, word_type := UInt, dword_type := UDInt, byte_type := USInt, any_type := Variant]" } "Modbus_Master_DB".Modbus_Master(REQ := wire#w1, MB_ADDR := 1, MODE := 0, DATA_ADDR := 32038, DATA_LEN := 1, DATA_PTR := "Modbus_Send_Receive_1".Reading_Struct."32038", DONE => "Modbus".Done, BUSY => "Modbus".Busy, ERROR => "Modbus".Error, STATUS => "Modbus".Status)
   END_RUNG
   RUNG wire#powerrail
      Contact( "Comm_ok" )
      { S7_Templates := "SrcType := Int" } EQ_Contact(in1 := "IEC_Counter_0_DB".CV, in2 := 32)
      I_Contact( "Modbus_Master_DB".BUSY )
   END_RUNG wire#w1
   // the same network as SCL:
   IF "IEC_Counter_0_DB".CV = 32 THEN
       "Modbus_Master_DB"(REQ := "Comm_ok" AND ("IEC_Counter_0_DB".CV = 32) AND NOT "Modbus_Master_DB".BUSY,   // Modbus_Master
                          MB_ADDR := 1,
                          MODE := 0,
                          DATA_ADDR := 32038,
                          DATA_LEN := 1,
                          DATA_PTR := "Modbus_Send_Receive_1".Reading_Struct."32038",
                          DONE => "Modbus".Done,
                          BUSY => "Modbus".Busy,
                          ERROR => "Modbus".Error,
                          STATUS => "Modbus".Status);
   END_IF;
END_REGION

REGION Network 38: RD 32039
   RUNG wire#powerrail
      { S7_Templates := "SrcType := Int" } EQ_Contact(in1 := "IEC_Counter_0_DB".CV, in2 := 33)
      { S7_Templates := "[card := 0, word_type := UInt, dword_type := UDInt, byte_type := USInt, any_type := Variant]" } "Modbus_Master_DB".Modbus_Master(REQ := wire#w1, MB_ADDR := 1, MODE := 0, DATA_ADDR := 32039, DATA_LEN := 1, DATA_PTR := "Modbus_Send_Receive_1".Reading_Struct."32039", DONE => "Modbus".Done, BUSY => "Modbus".Busy, ERROR => "Modbus".Error, STATUS => "Modbus".Status)
   END_RUNG
   RUNG wire#powerrail
      Contact( "Comm_ok" )
      { S7_Templates := "SrcType := Int" } EQ_Contact(in1 := "IEC_Counter_0_DB".CV, in2 := 33)
      I_Contact( "Modbus_Master_DB".BUSY )
   END_RUNG wire#w1
   // the same network as SCL:
   IF "IEC_Counter_0_DB".CV = 33 THEN
       "Modbus_Master_DB"(REQ := "Comm_ok" AND ("IEC_Counter_0_DB".CV = 33) AND NOT "Modbus_Master_DB".BUSY,   // Modbus_Master
                          MB_ADDR := 1,
                          MODE := 0,
                          DATA_ADDR := 32039,
                          DATA_LEN := 1,
                          DATA_PTR := "Modbus_Send_Receive_1".Reading_Struct."32039",
                          DONE => "Modbus".Done,
                          BUSY => "Modbus".Busy,
                          ERROR => "Modbus".Error,
                          STATUS => "Modbus".Status);
   END_IF;
END_REGION

REGION Network 39: RD 32040
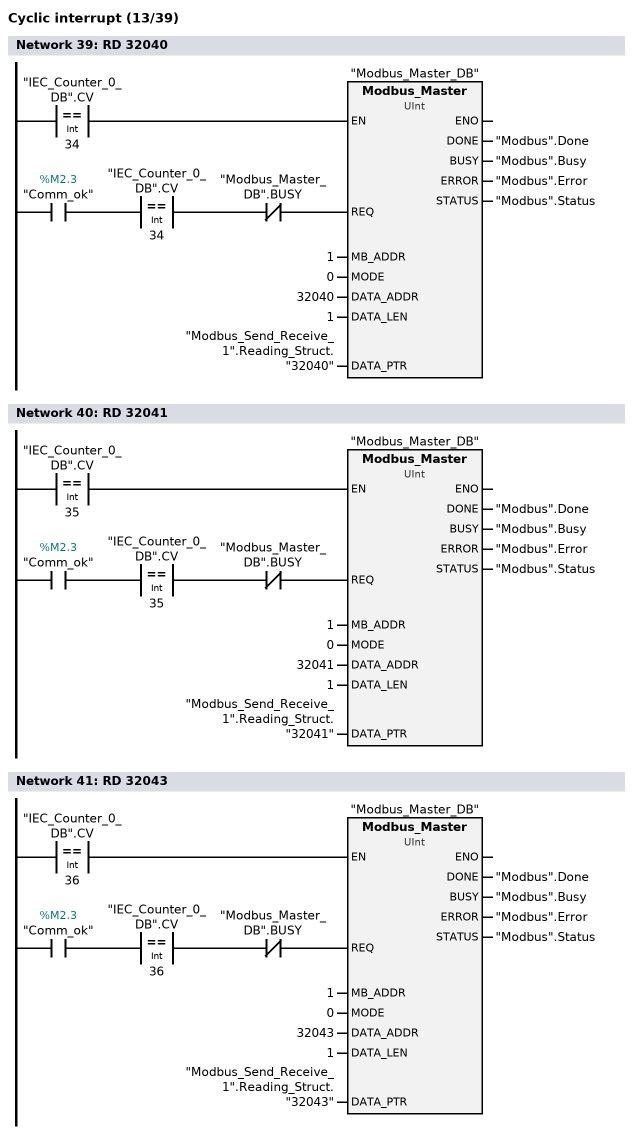
   RUNG wire#powerrail
      { S7_Templates := "SrcType := Int" } EQ_Contact(in1 := "IEC_Counter_0_DB".CV, in2 := 34)
      { S7_Templates := "[card := 0, word_type := UInt, dword_type := UDInt, byte_type := USInt, any_type := Variant]" } "Modbus_Master_DB".Modbus_Master(REQ := wire#w1, MB_ADDR := 1, MODE := 0, DATA_ADDR := 32040, DATA_LEN := 1, DATA_PTR := "Modbus_Send_Receive_1".Reading_Struct."32040", DONE => "Modbus".Done, BUSY => "Modbus".Busy, ERROR => "Modbus".Error, STATUS => "Modbus".Status)
   END_RUNG
   RUNG wire#powerrail
      Contact( "Comm_ok" )
      { S7_Templates := "SrcType := Int" } EQ_Contact(in1 := "IEC_Counter_0_DB".CV, in2 := 34)
      I_Contact( "Modbus_Master_DB".BUSY )
   END_RUNG wire#w1
   // the same network as SCL:
   IF "IEC_Counter_0_DB".CV = 34 THEN
       "Modbus_Master_DB"(REQ := "Comm_ok" AND ("IEC_Counter_0_DB".CV = 34) AND NOT "Modbus_Master_DB".BUSY,   // Modbus_Master
                          MB_ADDR := 1,
                          MODE := 0,
                          DATA_ADDR := 32040,
                          DATA_LEN := 1,
                          DATA_PTR := "Modbus_Send_Receive_1".Reading_Struct."32040",
                          DONE => "Modbus".Done,
                          BUSY => "Modbus".Busy,
                          ERROR => "Modbus".Error,
                          STATUS => "Modbus".Status);
   END_IF;
END_REGION

REGION Network 40: RD 32041
   RUNG wire#powerrail
      { S7_Templates := "SrcType := Int" } EQ_Contact(in1 := "IEC_Counter_0_DB".CV, in2 := 35)
      { S7_Templates := "[card := 0, word_type := UInt, dword_type := UDInt, byte_type := USInt, any_type := Variant]" } "Modbus_Master_DB".Modbus_Master(REQ := wire#w1, MB_ADDR := 1, MODE := 0, DATA_ADDR := 32041, DATA_LEN := 1, DATA_PTR := "Modbus_Send_Receive_1".Reading_Struct."32041", DONE => "Modbus".Done, BUSY => "Modbus".Busy, ERROR => "Modbus".Error, STATUS => "Modbus".Status)
   END_RUNG
   RUNG wire#powerrail
      Contact( "Comm_ok" )
      { S7_Templates := "SrcType := Int" } EQ_Contact(in1 := "IEC_Counter_0_DB".CV, in2 := 35)
      I_Contact( "Modbus_Master_DB".BUSY )
   END_RUNG wire#w1
   // the same network as SCL:
   IF "IEC_Counter_0_DB".CV = 35 THEN
       "Modbus_Master_DB"(REQ := "Comm_ok" AND ("IEC_Counter_0_DB".CV = 35) AND NOT "Modbus_Master_DB".BUSY,   // Modbus_Master
                          MB_ADDR := 1,
                          MODE := 0,
                          DATA_ADDR := 32041,
                          DATA_LEN := 1,
                          DATA_PTR := "Modbus_Send_Receive_1".Reading_Struct."32041",
                          DONE => "Modbus".Done,
                          BUSY => "Modbus".Busy,
                          ERROR => "Modbus".Error,
                          STATUS => "Modbus".Status);
   END_IF;
END_REGION

REGION Network 41: RD 32043
   RUNG wire#powerrail
      { S7_Templates := "SrcType := Int" } EQ_Contact(in1 := "IEC_Counter_0_DB".CV, in2 := 36)
      { S7_Templates := "[card := 0, word_type := UInt, dword_type := UDInt, byte_type := USInt, any_type := Variant]" } "Modbus_Master_DB".Modbus_Master(REQ := wire#w1, MB_ADDR := 1, MODE := 0, DATA_ADDR := 32043, DATA_LEN := 1, DATA_PTR := "Modbus_Send_Receive_1".Reading_Struct."32043", DONE => "Modbus".Done, BUSY => "Modbus".Busy, ERROR => "Modbus".Error, STATUS => "Modbus".Status)
   END_RUNG
   RUNG wire#powerrail
      Contact( "Comm_ok" )
      { S7_Templates := "SrcType := Int" } EQ_Contact(in1 := "IEC_Counter_0_DB".CV, in2 := 36)
      I_Contact( "Modbus_Master_DB".BUSY )
   END_RUNG wire#w1
   // the same network as SCL:
   IF "IEC_Counter_0_DB".CV = 36 THEN
       "Modbus_Master_DB"(REQ := "Comm_ok" AND ("IEC_Counter_0_DB".CV = 36) AND NOT "Modbus_Master_DB".BUSY,   // Modbus_Master
                          MB_ADDR := 1,
                          MODE := 0,
                          DATA_ADDR := 32043,
                          DATA_LEN := 1,
                          DATA_PTR := "Modbus_Send_Receive_1".Reading_Struct."32043",
                          DONE => "Modbus".Done,
                          BUSY => "Modbus".Busy,
                          ERROR => "Modbus".Error,
                          STATUS => "Modbus".Status);
   END_IF;
END_REGION

REGION Network 42: RD 32044
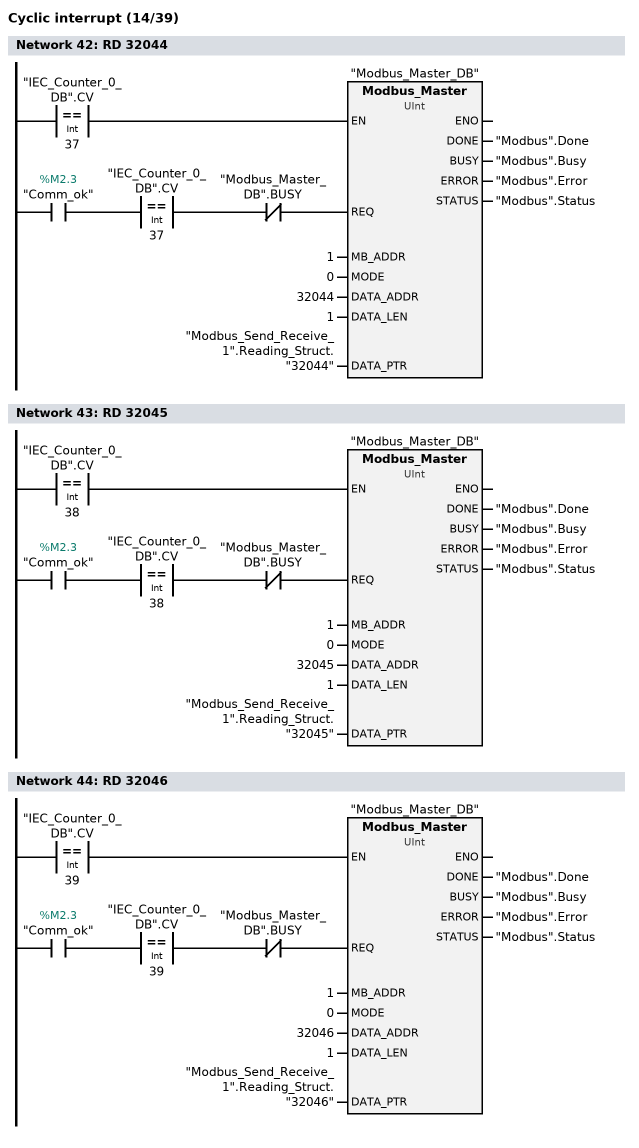
   RUNG wire#powerrail
      { S7_Templates := "SrcType := Int" } EQ_Contact(in1 := "IEC_Counter_0_DB".CV, in2 := 37)
      { S7_Templates := "[card := 0, word_type := UInt, dword_type := UDInt, byte_type := USInt, any_type := Variant]" } "Modbus_Master_DB".Modbus_Master(REQ := wire#w1, MB_ADDR := 1, MODE := 0, DATA_ADDR := 32044, DATA_LEN := 1, DATA_PTR := "Modbus_Send_Receive_1".Reading_Struct."32044", DONE => "Modbus".Done, BUSY => "Modbus".Busy, ERROR => "Modbus".Error, STATUS => "Modbus".Status)
   END_RUNG
   RUNG wire#powerrail
      Contact( "Comm_ok" )
      { S7_Templates := "SrcType := Int" } EQ_Contact(in1 := "IEC_Counter_0_DB".CV, in2 := 37)
      I_Contact( "Modbus_Master_DB".BUSY )
   END_RUNG wire#w1
   // the same network as SCL:
   IF "IEC_Counter_0_DB".CV = 37 THEN
       "Modbus_Master_DB"(REQ := "Comm_ok" AND ("IEC_Counter_0_DB".CV = 37) AND NOT "Modbus_Master_DB".BUSY,   // Modbus_Master
                          MB_ADDR := 1,
                          MODE := 0,
                          DATA_ADDR := 32044,
                          DATA_LEN := 1,
                          DATA_PTR := "Modbus_Send_Receive_1".Reading_Struct."32044",
                          DONE => "Modbus".Done,
                          BUSY => "Modbus".Busy,
                          ERROR => "Modbus".Error,
                          STATUS => "Modbus".Status);
   END_IF;
END_REGION

REGION Network 43: RD 32045
   RUNG wire#powerrail
      { S7_Templates := "SrcType := Int" } EQ_Contact(in1 := "IEC_Counter_0_DB".CV, in2 := 38)
      { S7_Templates := "[card := 0, word_type := UInt, dword_type := UDInt, byte_type := USInt, any_type := Variant]" } "Modbus_Master_DB".Modbus_Master(REQ := wire#w1, MB_ADDR := 1, MODE := 0, DATA_ADDR := 32045, DATA_LEN := 1, DATA_PTR := "Modbus_Send_Receive_1".Reading_Struct."32045", DONE => "Modbus".Done, BUSY => "Modbus".Busy, ERROR => "Modbus".Error, STATUS => "Modbus".Status)
   END_RUNG
   RUNG wire#powerrail
      Contact( "Comm_ok" )
      { S7_Templates := "SrcType := Int" } EQ_Contact(in1 := "IEC_Counter_0_DB".CV, in2 := 38)
      I_Contact( "Modbus_Master_DB".BUSY )
   END_RUNG wire#w1
   // the same network as SCL:
   IF "IEC_Counter_0_DB".CV = 38 THEN
       "Modbus_Master_DB"(REQ := "Comm_ok" AND ("IEC_Counter_0_DB".CV = 38) AND NOT "Modbus_Master_DB".BUSY,   // Modbus_Master
                          MB_ADDR := 1,
                          MODE := 0,
                          DATA_ADDR := 32045,
                          DATA_LEN := 1,
                          DATA_PTR := "Modbus_Send_Receive_1".Reading_Struct."32045",
                          DONE => "Modbus".Done,
                          BUSY => "Modbus".Busy,
                          ERROR => "Modbus".Error,
                          STATUS => "Modbus".Status);
   END_IF;
END_REGION

REGION Network 44: RD 32046
   RUNG wire#powerrail
      { S7_Templates := "SrcType := Int" } EQ_Contact(in1 := "IEC_Counter_0_DB".CV, in2 := 39)
      { S7_Templates := "[card := 0, word_type := UInt, dword_type := UDInt, byte_type := USInt, any_type := Variant]" } "Modbus_Master_DB".Modbus_Master(REQ := wire#w1, MB_ADDR := 1, MODE := 0, DATA_ADDR := 32046, DATA_LEN := 1, DATA_PTR := "Modbus_Send_Receive_1".Reading_Struct."32046", DONE => "Modbus".Done, BUSY => "Modbus".Busy, ERROR => "Modbus".Error, STATUS => "Modbus".Status)
   END_RUNG
   RUNG wire#powerrail
      Contact( "Comm_ok" )
      { S7_Templates := "SrcType := Int" } EQ_Contact(in1 := "IEC_Counter_0_DB".CV, in2 := 39)
      I_Contact( "Modbus_Master_DB".BUSY )
   END_RUNG wire#w1
   // the same network as SCL:
   IF "IEC_Counter_0_DB".CV = 39 THEN
       "Modbus_Master_DB"(REQ := "Comm_ok" AND ("IEC_Counter_0_DB".CV = 39) AND NOT "Modbus_Master_DB".BUSY,   // Modbus_Master
                          MB_ADDR := 1,
                          MODE := 0,
                          DATA_ADDR := 32046,
                          DATA_LEN := 1,
                          DATA_PTR := "Modbus_Send_Receive_1".Reading_Struct."32046",
                          DONE => "Modbus".Done,
                          BUSY => "Modbus".Busy,
                          ERROR => "Modbus".Error,
                          STATUS => "Modbus".Status);
   END_IF;
END_REGION

REGION Network 45: RD 32047
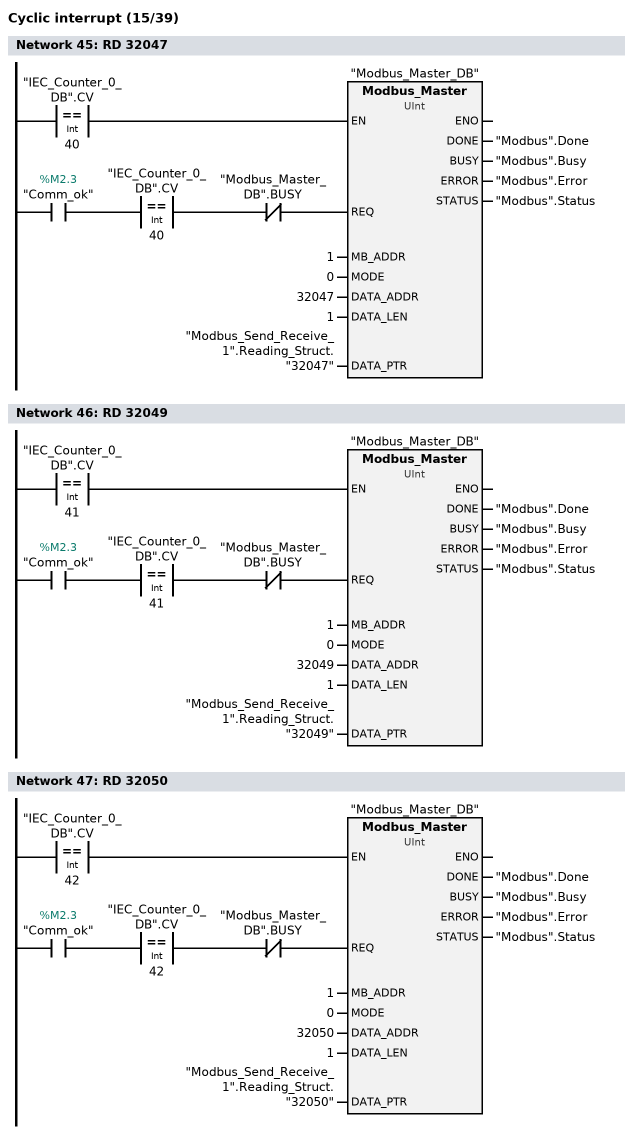
   RUNG wire#powerrail
      { S7_Templates := "SrcType := Int" } EQ_Contact(in1 := "IEC_Counter_0_DB".CV, in2 := 40)
      { S7_Templates := "[card := 0, word_type := UInt, dword_type := UDInt, byte_type := USInt, any_type := Variant]" } "Modbus_Master_DB".Modbus_Master(REQ := wire#w1, MB_ADDR := 1, MODE := 0, DATA_ADDR := 32047, DATA_LEN := 1, DATA_PTR := "Modbus_Send_Receive_1".Reading_Struct."32047", DONE => "Modbus".Done, BUSY => "Modbus".Busy, ERROR => "Modbus".Error, STATUS => "Modbus".Status)
   END_RUNG
   RUNG wire#powerrail
      Contact( "Comm_ok" )
      { S7_Templates := "SrcType := Int" } EQ_Contact(in1 := "IEC_Counter_0_DB".CV, in2 := 40)
      I_Contact( "Modbus_Master_DB".BUSY )
   END_RUNG wire#w1
   // the same network as SCL:
   IF "IEC_Counter_0_DB".CV = 40 THEN
       "Modbus_Master_DB"(REQ := "Comm_ok" AND ("IEC_Counter_0_DB".CV = 40) AND NOT "Modbus_Master_DB".BUSY,   // Modbus_Master
                          MB_ADDR := 1,
                          MODE := 0,
                          DATA_ADDR := 32047,
                          DATA_LEN := 1,
                          DATA_PTR := "Modbus_Send_Receive_1".Reading_Struct."32047",
                          DONE => "Modbus".Done,
                          BUSY => "Modbus".Busy,
                          ERROR => "Modbus".Error,
                          STATUS => "Modbus".Status);
   END_IF;
END_REGION

REGION Network 46: RD 32049
   RUNG wire#powerrail
      { S7_Templates := "SrcType := Int" } EQ_Contact(in1 := "IEC_Counter_0_DB".CV, in2 := 41)
      { S7_Templates := "[card := 0, word_type := UInt, dword_type := UDInt, byte_type := USInt, any_type := Variant]" } "Modbus_Master_DB".Modbus_Master(REQ := wire#w1, MB_ADDR := 1, MODE := 0, DATA_ADDR := 32049, DATA_LEN := 1, DATA_PTR := "Modbus_Send_Receive_1".Reading_Struct."32049", DONE => "Modbus".Done, BUSY => "Modbus".Busy, ERROR => "Modbus".Error, STATUS => "Modbus".Status)
   END_RUNG
   RUNG wire#powerrail
      Contact( "Comm_ok" )
      { S7_Templates := "SrcType := Int" } EQ_Contact(in1 := "IEC_Counter_0_DB".CV, in2 := 41)
      I_Contact( "Modbus_Master_DB".BUSY )
   END_RUNG wire#w1
   // the same network as SCL:
   IF "IEC_Counter_0_DB".CV = 41 THEN
       "Modbus_Master_DB"(REQ := "Comm_ok" AND ("IEC_Counter_0_DB".CV = 41) AND NOT "Modbus_Master_DB".BUSY,   // Modbus_Master
                          MB_ADDR := 1,
                          MODE := 0,
                          DATA_ADDR := 32049,
                          DATA_LEN := 1,
                          DATA_PTR := "Modbus_Send_Receive_1".Reading_Struct."32049",
                          DONE => "Modbus".Done,
                          BUSY => "Modbus".Busy,
                          ERROR => "Modbus".Error,
                          STATUS => "Modbus".Status);
   END_IF;
END_REGION

REGION Network 47: RD 32050
   RUNG wire#powerrail
      { S7_Templates := "SrcType := Int" } EQ_Contact(in1 := "IEC_Counter_0_DB".CV, in2 := 42)
      { S7_Templates := "[card := 0, word_type := UInt, dword_type := UDInt, byte_type := USInt, any_type := Variant]" } "Modbus_Master_DB".Modbus_Master(REQ := wire#w1, MB_ADDR := 1, MODE := 0, DATA_ADDR := 32050, DATA_LEN := 1, DATA_PTR := "Modbus_Send_Receive_1".Reading_Struct."32050", DONE => "Modbus".Done, BUSY => "Modbus".Busy, ERROR => "Modbus".Error, STATUS => "Modbus".Status)
   END_RUNG
   RUNG wire#powerrail
      Contact( "Comm_ok" )
      { S7_Templates := "SrcType := Int" } EQ_Contact(in1 := "IEC_Counter_0_DB".CV, in2 := 42)
      I_Contact( "Modbus_Master_DB".BUSY )
   END_RUNG wire#w1
   // the same network as SCL:
   IF "IEC_Counter_0_DB".CV = 42 THEN
       "Modbus_Master_DB"(REQ := "Comm_ok" AND ("IEC_Counter_0_DB".CV = 42) AND NOT "Modbus_Master_DB".BUSY,   // Modbus_Master
                          MB_ADDR := 1,
                          MODE := 0,
                          DATA_ADDR := 32050,
                          DATA_LEN := 1,
                          DATA_PTR := "Modbus_Send_Receive_1".Reading_Struct."32050",
                          DONE => "Modbus".Done,
                          BUSY => "Modbus".Busy,
                          ERROR => "Modbus".Error,
                          STATUS => "Modbus".Status);
   END_IF;
END_REGION

REGION Network 48: RD 32051
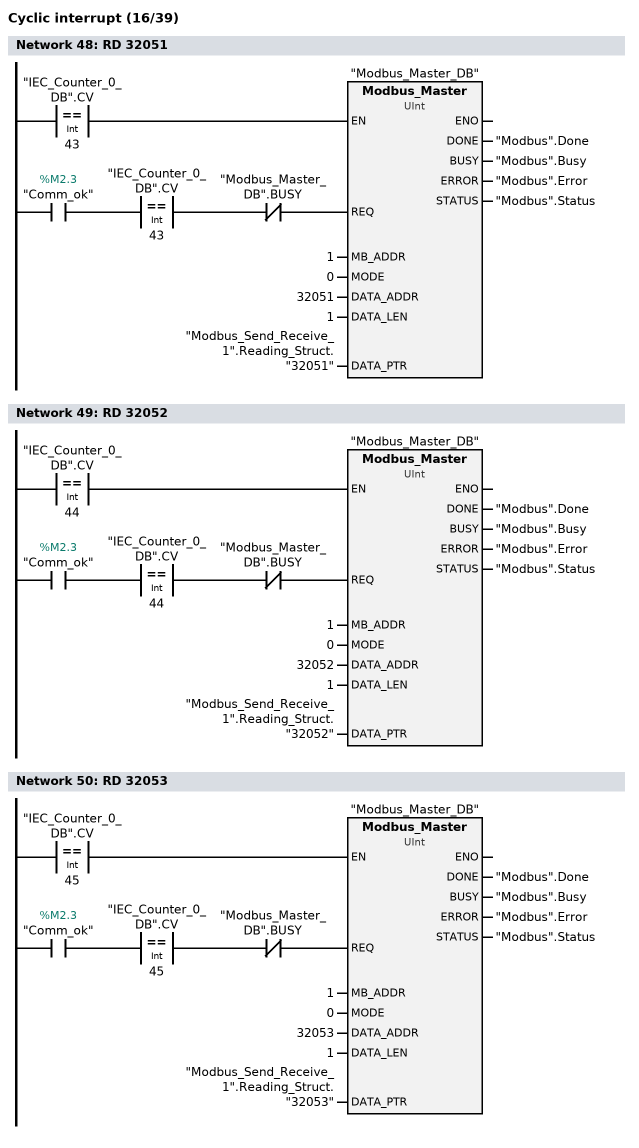
   RUNG wire#powerrail
      { S7_Templates := "SrcType := Int" } EQ_Contact(in1 := "IEC_Counter_0_DB".CV, in2 := 43)
      { S7_Templates := "[card := 0, word_type := UInt, dword_type := UDInt, byte_type := USInt, any_type := Variant]" } "Modbus_Master_DB".Modbus_Master(REQ := wire#w1, MB_ADDR := 1, MODE := 0, DATA_ADDR := 32051, DATA_LEN := 1, DATA_PTR := "Modbus_Send_Receive_1".Reading_Struct."32051", DONE => "Modbus".Done, BUSY => "Modbus".Busy, ERROR => "Modbus".Error, STATUS => "Modbus".Status)
   END_RUNG
   RUNG wire#powerrail
      Contact( "Comm_ok" )
      { S7_Templates := "SrcType := Int" } EQ_Contact(in1 := "IEC_Counter_0_DB".CV, in2 := 43)
      I_Contact( "Modbus_Master_DB".BUSY )
   END_RUNG wire#w1
   // the same network as SCL:
   IF "IEC_Counter_0_DB".CV = 43 THEN
       "Modbus_Master_DB"(REQ := "Comm_ok" AND ("IEC_Counter_0_DB".CV = 43) AND NOT "Modbus_Master_DB".BUSY,   // Modbus_Master
                          MB_ADDR := 1,
                          MODE := 0,
                          DATA_ADDR := 32051,
                          DATA_LEN := 1,
                          DATA_PTR := "Modbus_Send_Receive_1".Reading_Struct."32051",
                          DONE => "Modbus".Done,
                          BUSY => "Modbus".Busy,
                          ERROR => "Modbus".Error,
                          STATUS => "Modbus".Status);
   END_IF;
END_REGION

REGION Network 49: RD 32052
   RUNG wire#powerrail
      { S7_Templates := "SrcType := Int" } EQ_Contact(in1 := "IEC_Counter_0_DB".CV, in2 := 44)
      { S7_Templates := "[card := 0, word_type := UInt, dword_type := UDInt, byte_type := USInt, any_type := Variant]" } "Modbus_Master_DB".Modbus_Master(REQ := wire#w1, MB_ADDR := 1, MODE := 0, DATA_ADDR := 32052, DATA_LEN := 1, DATA_PTR := "Modbus_Send_Receive_1".Reading_Struct."32052", DONE => "Modbus".Done, BUSY => "Modbus".Busy, ERROR => "Modbus".Error, STATUS => "Modbus".Status)
   END_RUNG
   RUNG wire#powerrail
      Contact( "Comm_ok" )
      { S7_Templates := "SrcType := Int" } EQ_Contact(in1 := "IEC_Counter_0_DB".CV, in2 := 44)
      I_Contact( "Modbus_Master_DB".BUSY )
   END_RUNG wire#w1
   // the same network as SCL:
   IF "IEC_Counter_0_DB".CV = 44 THEN
       "Modbus_Master_DB"(REQ := "Comm_ok" AND ("IEC_Counter_0_DB".CV = 44) AND NOT "Modbus_Master_DB".BUSY,   // Modbus_Master
                          MB_ADDR := 1,
                          MODE := 0,
                          DATA_ADDR := 32052,
                          DATA_LEN := 1,
                          DATA_PTR := "Modbus_Send_Receive_1".Reading_Struct."32052",
                          DONE => "Modbus".Done,
                          BUSY => "Modbus".Busy,
                          ERROR => "Modbus".Error,
                          STATUS => "Modbus".Status);
   END_IF;
END_REGION

REGION Network 50: RD 32053
   RUNG wire#powerrail
      { S7_Templates := "SrcType := Int" } EQ_Contact(in1 := "IEC_Counter_0_DB".CV, in2 := 45)
      { S7_Templates := "[card := 0, word_type := UInt, dword_type := UDInt, byte_type := USInt, any_type := Variant]" } "Modbus_Master_DB".Modbus_Master(REQ := wire#w1, MB_ADDR := 1, MODE := 0, DATA_ADDR := 32053, DATA_LEN := 1, DATA_PTR := "Modbus_Send_Receive_1".Reading_Struct."32053", DONE => "Modbus".Done, BUSY => "Modbus".Busy, ERROR => "Modbus".Error, STATUS => "Modbus".Status)
   END_RUNG
   RUNG wire#powerrail
      Contact( "Comm_ok" )
      { S7_Templates := "SrcType := Int" } EQ_Contact(in1 := "IEC_Counter_0_DB".CV, in2 := 45)
      I_Contact( "Modbus_Master_DB".BUSY )
   END_RUNG wire#w1
   // the same network as SCL:
   IF "IEC_Counter_0_DB".CV = 45 THEN
       "Modbus_Master_DB"(REQ := "Comm_ok" AND ("IEC_Counter_0_DB".CV = 45) AND NOT "Modbus_Master_DB".BUSY,   // Modbus_Master
                          MB_ADDR := 1,
                          MODE := 0,
                          DATA_ADDR := 32053,
                          DATA_LEN := 1,
                          DATA_PTR := "Modbus_Send_Receive_1".Reading_Struct."32053",
                          DONE => "Modbus".Done,
                          BUSY => "Modbus".Busy,
                          ERROR => "Modbus".Error,
                          STATUS => "Modbus".Status);
   END_IF;
END_REGION

REGION Network 51: RD 32055
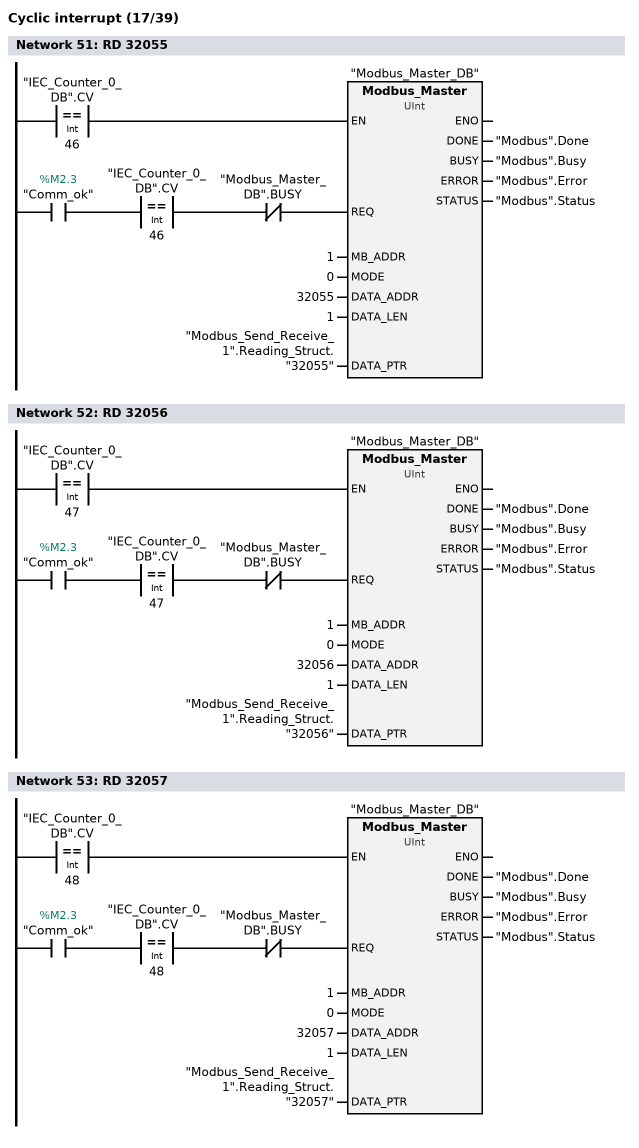
   RUNG wire#powerrail
      { S7_Templates := "SrcType := Int" } EQ_Contact(in1 := "IEC_Counter_0_DB".CV, in2 := 46)
      { S7_Templates := "[card := 0, word_type := UInt, dword_type := UDInt, byte_type := USInt, any_type := Variant]" } "Modbus_Master_DB".Modbus_Master(REQ := wire#w1, MB_ADDR := 1, MODE := 0, DATA_ADDR := 32055, DATA_LEN := 1, DATA_PTR := "Modbus_Send_Receive_1".Reading_Struct."32055", DONE => "Modbus".Done, BUSY => "Modbus".Busy, ERROR => "Modbus".Error, STATUS => "Modbus".Status)
   END_RUNG
   RUNG wire#powerrail
      Contact( "Comm_ok" )
      { S7_Templates := "SrcType := Int" } EQ_Contact(in1 := "IEC_Counter_0_DB".CV, in2 := 46)
      I_Contact( "Modbus_Master_DB".BUSY )
   END_RUNG wire#w1
   // the same network as SCL:
   IF "IEC_Counter_0_DB".CV = 46 THEN
       "Modbus_Master_DB"(REQ := "Comm_ok" AND ("IEC_Counter_0_DB".CV = 46) AND NOT "Modbus_Master_DB".BUSY,   // Modbus_Master
                          MB_ADDR := 1,
                          MODE := 0,
                          DATA_ADDR := 32055,
                          DATA_LEN := 1,
                          DATA_PTR := "Modbus_Send_Receive_1".Reading_Struct."32055",
                          DONE => "Modbus".Done,
                          BUSY => "Modbus".Busy,
                          ERROR => "Modbus".Error,
                          STATUS => "Modbus".Status);
   END_IF;
END_REGION

REGION Network 52: RD 32056
   RUNG wire#powerrail
      { S7_Templates := "SrcType := Int" } EQ_Contact(in1 := "IEC_Counter_0_DB".CV, in2 := 47)
      { S7_Templates := "[card := 0, word_type := UInt, dword_type := UDInt, byte_type := USInt, any_type := Variant]" } "Modbus_Master_DB".Modbus_Master(REQ := wire#w1, MB_ADDR := 1, MODE := 0, DATA_ADDR := 32056, DATA_LEN := 1, DATA_PTR := "Modbus_Send_Receive_1".Reading_Struct."32056", DONE => "Modbus".Done, BUSY => "Modbus".Busy, ERROR => "Modbus".Error, STATUS => "Modbus".Status)
   END_RUNG
   RUNG wire#powerrail
      Contact( "Comm_ok" )
      { S7_Templates := "SrcType := Int" } EQ_Contact(in1 := "IEC_Counter_0_DB".CV, in2 := 47)
      I_Contact( "Modbus_Master_DB".BUSY )
   END_RUNG wire#w1
   // the same network as SCL:
   IF "IEC_Counter_0_DB".CV = 47 THEN
       "Modbus_Master_DB"(REQ := "Comm_ok" AND ("IEC_Counter_0_DB".CV = 47) AND NOT "Modbus_Master_DB".BUSY,   // Modbus_Master
                          MB_ADDR := 1,
                          MODE := 0,
                          DATA_ADDR := 32056,
                          DATA_LEN := 1,
                          DATA_PTR := "Modbus_Send_Receive_1".Reading_Struct."32056",
                          DONE => "Modbus".Done,
                          BUSY => "Modbus".Busy,
                          ERROR => "Modbus".Error,
                          STATUS => "Modbus".Status);
   END_IF;
END_REGION

REGION Network 53: RD 32057
   RUNG wire#powerrail
      { S7_Templates := "SrcType := Int" } EQ_Contact(in1 := "IEC_Counter_0_DB".CV, in2 := 48)
      { S7_Templates := "[card := 0, word_type := UInt, dword_type := UDInt, byte_type := USInt, any_type := Variant]" } "Modbus_Master_DB".Modbus_Master(REQ := wire#w1, MB_ADDR := 1, MODE := 0, DATA_ADDR := 32057, DATA_LEN := 1, DATA_PTR := "Modbus_Send_Receive_1".Reading_Struct."32057", DONE => "Modbus".Done, BUSY => "Modbus".Busy, ERROR => "Modbus".Error, STATUS => "Modbus".Status)
   END_RUNG
   RUNG wire#powerrail
      Contact( "Comm_ok" )
      { S7_Templates := "SrcType := Int" } EQ_Contact(in1 := "IEC_Counter_0_DB".CV, in2 := 48)
      I_Contact( "Modbus_Master_DB".BUSY )
   END_RUNG wire#w1
   // the same network as SCL:
   IF "IEC_Counter_0_DB".CV = 48 THEN
       "Modbus_Master_DB"(REQ := "Comm_ok" AND ("IEC_Counter_0_DB".CV = 48) AND NOT "Modbus_Master_DB".BUSY,   // Modbus_Master
                          MB_ADDR := 1,
                          MODE := 0,
                          DATA_ADDR := 32057,
                          DATA_LEN := 1,
                          DATA_PTR := "Modbus_Send_Receive_1".Reading_Struct."32057",
                          DONE => "Modbus".Done,
                          BUSY => "Modbus".Busy,
                          ERROR => "Modbus".Error,
                          STATUS => "Modbus".Status);
   END_IF;
END_REGION

REGION Network 54: RD 32058
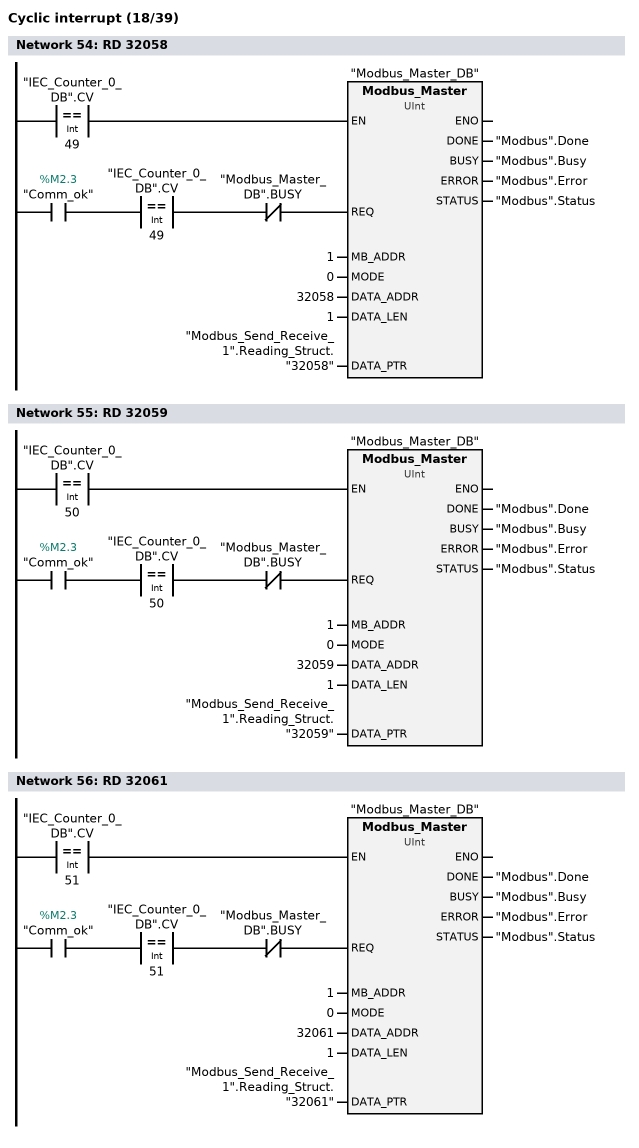
   RUNG wire#powerrail
      { S7_Templates := "SrcType := Int" } EQ_Contact(in1 := "IEC_Counter_0_DB".CV, in2 := 49)
      { S7_Templates := "[card := 0, word_type := UInt, dword_type := UDInt, byte_type := USInt, any_type := Variant]" } "Modbus_Master_DB".Modbus_Master(REQ := wire#w1, MB_ADDR := 1, MODE := 0, DATA_ADDR := 32058, DATA_LEN := 1, DATA_PTR := "Modbus_Send_Receive_1".Reading_Struct."32058", DONE => "Modbus".Done, BUSY => "Modbus".Busy, ERROR => "Modbus".Error, STATUS => "Modbus".Status)
   END_RUNG
   RUNG wire#powerrail
      Contact( "Comm_ok" )
      { S7_Templates := "SrcType := Int" } EQ_Contact(in1 := "IEC_Counter_0_DB".CV, in2 := 49)
      I_Contact( "Modbus_Master_DB".BUSY )
   END_RUNG wire#w1
   // the same network as SCL:
   IF "IEC_Counter_0_DB".CV = 49 THEN
       "Modbus_Master_DB"(REQ := "Comm_ok" AND ("IEC_Counter_0_DB".CV = 49) AND NOT "Modbus_Master_DB".BUSY,   // Modbus_Master
                          MB_ADDR := 1,
                          MODE := 0,
                          DATA_ADDR := 32058,
                          DATA_LEN := 1,
                          DATA_PTR := "Modbus_Send_Receive_1".Reading_Struct."32058",
                          DONE => "Modbus".Done,
                          BUSY => "Modbus".Busy,
                          ERROR => "Modbus".Error,
                          STATUS => "Modbus".Status);
   END_IF;
END_REGION

REGION Network 55: RD 32059
   RUNG wire#powerrail
      { S7_Templates := "SrcType := Int" } EQ_Contact(in1 := "IEC_Counter_0_DB".CV, in2 := 50)
      { S7_Templates := "[card := 0, word_type := UInt, dword_type := UDInt, byte_type := USInt, any_type := Variant]" } "Modbus_Master_DB".Modbus_Master(REQ := wire#w1, MB_ADDR := 1, MODE := 0, DATA_ADDR := 32059, DATA_LEN := 1, DATA_PTR := "Modbus_Send_Receive_1".Reading_Struct."32059", DONE => "Modbus".Done, BUSY => "Modbus".Busy, ERROR => "Modbus".Error, STATUS => "Modbus".Status)
   END_RUNG
   RUNG wire#powerrail
      Contact( "Comm_ok" )
      { S7_Templates := "SrcType := Int" } EQ_Contact(in1 := "IEC_Counter_0_DB".CV, in2 := 50)
      I_Contact( "Modbus_Master_DB".BUSY )
   END_RUNG wire#w1
   // the same network as SCL:
   IF "IEC_Counter_0_DB".CV = 50 THEN
       "Modbus_Master_DB"(REQ := "Comm_ok" AND ("IEC_Counter_0_DB".CV = 50) AND NOT "Modbus_Master_DB".BUSY,   // Modbus_Master
                          MB_ADDR := 1,
                          MODE := 0,
                          DATA_ADDR := 32059,
                          DATA_LEN := 1,
                          DATA_PTR := "Modbus_Send_Receive_1".Reading_Struct."32059",
                          DONE => "Modbus".Done,
                          BUSY => "Modbus".Busy,
                          ERROR => "Modbus".Error,
                          STATUS => "Modbus".Status);
   END_IF;
END_REGION

REGION Network 56: RD 32061
   RUNG wire#powerrail
      { S7_Templates := "SrcType := Int" } EQ_Contact(in1 := "IEC_Counter_0_DB".CV, in2 := 51)
      { S7_Templates := "[card := 0, word_type := UInt, dword_type := UDInt, byte_type := USInt, any_type := Variant]" } "Modbus_Master_DB".Modbus_Master(REQ := wire#w1, MB_ADDR := 1, MODE := 0, DATA_ADDR := 32061, DATA_LEN := 1, DATA_PTR := "Modbus_Send_Receive_1".Reading_Struct."32061", DONE => "Modbus".Done, BUSY => "Modbus".Busy, ERROR => "Modbus".Error, STATUS => "Modbus".Status)
   END_RUNG
   RUNG wire#powerrail
      Contact( "Comm_ok" )
      { S7_Templates := "SrcType := Int" } EQ_Contact(in1 := "IEC_Counter_0_DB".CV, in2 := 51)
      I_Contact( "Modbus_Master_DB".BUSY )
   END_RUNG wire#w1
   // the same network as SCL:
   IF "IEC_Counter_0_DB".CV = 51 THEN
       "Modbus_Master_DB"(REQ := "Comm_ok" AND ("IEC_Counter_0_DB".CV = 51) AND NOT "Modbus_Master_DB".BUSY,   // Modbus_Master
                          MB_ADDR := 1,
                          MODE := 0,
                          DATA_ADDR := 32061,
                          DATA_LEN := 1,
                          DATA_PTR := "Modbus_Send_Receive_1".Reading_Struct."32061",
                          DONE => "Modbus".Done,
                          BUSY => "Modbus".Busy,
                          ERROR => "Modbus".Error,
                          STATUS => "Modbus".Status);
   END_IF;
END_REGION

REGION Network 57: RD 32062
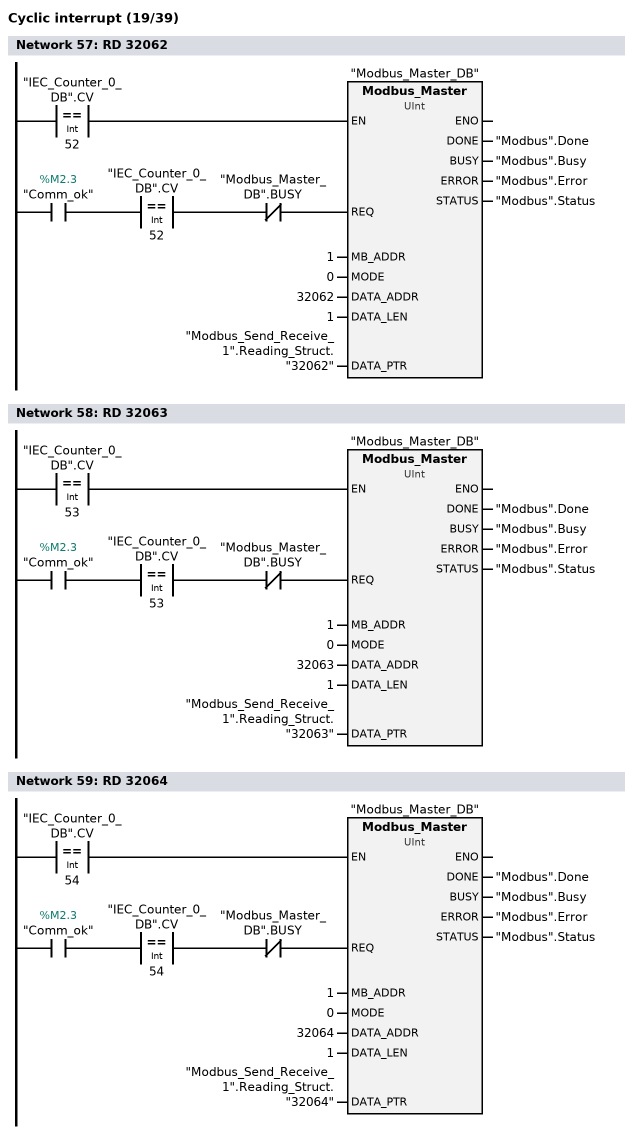
   RUNG wire#powerrail
      { S7_Templates := "SrcType := Int" } EQ_Contact(in1 := "IEC_Counter_0_DB".CV, in2 := 52)
      { S7_Templates := "[card := 0, word_type := UInt, dword_type := UDInt, byte_type := USInt, any_type := Variant]" } "Modbus_Master_DB".Modbus_Master(REQ := wire#w1, MB_ADDR := 1, MODE := 0, DATA_ADDR := 32062, DATA_LEN := 1, DATA_PTR := "Modbus_Send_Receive_1".Reading_Struct."32062", DONE => "Modbus".Done, BUSY => "Modbus".Busy, ERROR => "Modbus".Error, STATUS => "Modbus".Status)
   END_RUNG
   RUNG wire#powerrail
      Contact( "Comm_ok" )
      { S7_Templates := "SrcType := Int" } EQ_Contact(in1 := "IEC_Counter_0_DB".CV, in2 := 52)
      I_Contact( "Modbus_Master_DB".BUSY )
   END_RUNG wire#w1
   // the same network as SCL:
   IF "IEC_Counter_0_DB".CV = 52 THEN
       "Modbus_Master_DB"(REQ := "Comm_ok" AND ("IEC_Counter_0_DB".CV = 52) AND NOT "Modbus_Master_DB".BUSY,   // Modbus_Master
                          MB_ADDR := 1,
                          MODE := 0,
                          DATA_ADDR := 32062,
                          DATA_LEN := 1,
                          DATA_PTR := "Modbus_Send_Receive_1".Reading_Struct."32062",
                          DONE => "Modbus".Done,
                          BUSY => "Modbus".Busy,
                          ERROR => "Modbus".Error,
                          STATUS => "Modbus".Status);
   END_IF;
END_REGION

REGION Network 58: RD 32063
   RUNG wire#powerrail
      { S7_Templates := "SrcType := Int" } EQ_Contact(in1 := "IEC_Counter_0_DB".CV, in2 := 53)
      { S7_Templates := "[card := 0, word_type := UInt, dword_type := UDInt, byte_type := USInt, any_type := Variant]" } "Modbus_Master_DB".Modbus_Master(REQ := wire#w1, MB_ADDR := 1, MODE := 0, DATA_ADDR := 32063, DATA_LEN := 1, DATA_PTR := "Modbus_Send_Receive_1".Reading_Struct."32063", DONE => "Modbus".Done, BUSY => "Modbus".Busy, ERROR => "Modbus".Error, STATUS => "Modbus".Status)
   END_RUNG
   RUNG wire#powerrail
      Contact( "Comm_ok" )
      { S7_Templates := "SrcType := Int" } EQ_Contact(in1 := "IEC_Counter_0_DB".CV, in2 := 53)
      I_Contact( "Modbus_Master_DB".BUSY )
   END_RUNG wire#w1
   // the same network as SCL:
   IF "IEC_Counter_0_DB".CV = 53 THEN
       "Modbus_Master_DB"(REQ := "Comm_ok" AND ("IEC_Counter_0_DB".CV = 53) AND NOT "Modbus_Master_DB".BUSY,   // Modbus_Master
                          MB_ADDR := 1,
                          MODE := 0,
                          DATA_ADDR := 32063,
                          DATA_LEN := 1,
                          DATA_PTR := "Modbus_Send_Receive_1".Reading_Struct."32063",
                          DONE => "Modbus".Done,
                          BUSY => "Modbus".Busy,
                          ERROR => "Modbus".Error,
                          STATUS => "Modbus".Status);
   END_IF;
END_REGION

REGION Network 59: RD 32064
   RUNG wire#powerrail
      { S7_Templates := "SrcType := Int" } EQ_Contact(in1 := "IEC_Counter_0_DB".CV, in2 := 54)
      { S7_Templates := "[card := 0, word_type := UInt, dword_type := UDInt, byte_type := USInt, any_type := Variant]" } "Modbus_Master_DB".Modbus_Master(REQ := wire#w1, MB_ADDR := 1, MODE := 0, DATA_ADDR := 32064, DATA_LEN := 1, DATA_PTR := "Modbus_Send_Receive_1".Reading_Struct."32064", DONE => "Modbus".Done, BUSY => "Modbus".Busy, ERROR => "Modbus".Error, STATUS => "Modbus".Status)
   END_RUNG
   RUNG wire#powerrail
      Contact( "Comm_ok" )
      { S7_Templates := "SrcType := Int" } EQ_Contact(in1 := "IEC_Counter_0_DB".CV, in2 := 54)
      I_Contact( "Modbus_Master_DB".BUSY )
   END_RUNG wire#w1
   // the same network as SCL:
   IF "IEC_Counter_0_DB".CV = 54 THEN
       "Modbus_Master_DB"(REQ := "Comm_ok" AND ("IEC_Counter_0_DB".CV = 54) AND NOT "Modbus_Master_DB".BUSY,   // Modbus_Master
                          MB_ADDR := 1,
                          MODE := 0,
                          DATA_ADDR := 32064,
                          DATA_LEN := 1,
                          DATA_PTR := "Modbus_Send_Receive_1".Reading_Struct."32064",
                          DONE => "Modbus".Done,
                          BUSY => "Modbus".Busy,
                          ERROR => "Modbus".Error,
                          STATUS => "Modbus".Status);
   END_IF;
END_REGION

REGION Network 60: RD 32065
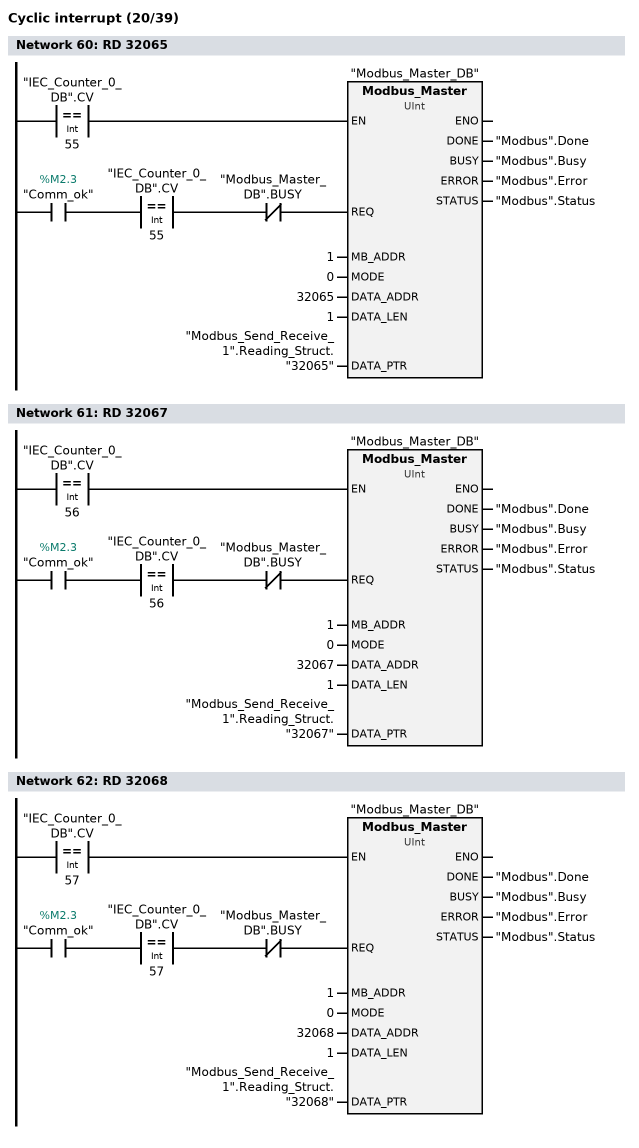
   RUNG wire#powerrail
      { S7_Templates := "SrcType := Int" } EQ_Contact(in1 := "IEC_Counter_0_DB".CV, in2 := 55)
      { S7_Templates := "[card := 0, word_type := UInt, dword_type := UDInt, byte_type := USInt, any_type := Variant]" } "Modbus_Master_DB".Modbus_Master(REQ := wire#w1, MB_ADDR := 1, MODE := 0, DATA_ADDR := 32065, DATA_LEN := 1, DATA_PTR := "Modbus_Send_Receive_1".Reading_Struct."32065", DONE => "Modbus".Done, BUSY => "Modbus".Busy, ERROR => "Modbus".Error, STATUS => "Modbus".Status)
   END_RUNG
   RUNG wire#powerrail
      Contact( "Comm_ok" )
      { S7_Templates := "SrcType := Int" } EQ_Contact(in1 := "IEC_Counter_0_DB".CV, in2 := 55)
      I_Contact( "Modbus_Master_DB".BUSY )
   END_RUNG wire#w1
   // the same network as SCL:
   IF "IEC_Counter_0_DB".CV = 55 THEN
       "Modbus_Master_DB"(REQ := "Comm_ok" AND ("IEC_Counter_0_DB".CV = 55) AND NOT "Modbus_Master_DB".BUSY,   // Modbus_Master
                          MB_ADDR := 1,
                          MODE := 0,
                          DATA_ADDR := 32065,
                          DATA_LEN := 1,
                          DATA_PTR := "Modbus_Send_Receive_1".Reading_Struct."32065",
                          DONE => "Modbus".Done,
                          BUSY => "Modbus".Busy,
                          ERROR => "Modbus".Error,
                          STATUS => "Modbus".Status);
   END_IF;
END_REGION

REGION Network 61: RD 32067
   RUNG wire#powerrail
      { S7_Templates := "SrcType := Int" } EQ_Contact(in1 := "IEC_Counter_0_DB".CV, in2 := 56)
      { S7_Templates := "[card := 0, word_type := UInt, dword_type := UDInt, byte_type := USInt, any_type := Variant]" } "Modbus_Master_DB".Modbus_Master(REQ := wire#w1, MB_ADDR := 1, MODE := 0, DATA_ADDR := 32067, DATA_LEN := 1, DATA_PTR := "Modbus_Send_Receive_1".Reading_Struct."32067", DONE => "Modbus".Done, BUSY => "Modbus".Busy, ERROR => "Modbus".Error, STATUS => "Modbus".Status)
   END_RUNG
   RUNG wire#powerrail
      Contact( "Comm_ok" )
      { S7_Templates := "SrcType := Int" } EQ_Contact(in1 := "IEC_Counter_0_DB".CV, in2 := 56)
      I_Contact( "Modbus_Master_DB".BUSY )
   END_RUNG wire#w1
   // the same network as SCL:
   IF "IEC_Counter_0_DB".CV = 56 THEN
       "Modbus_Master_DB"(REQ := "Comm_ok" AND ("IEC_Counter_0_DB".CV = 56) AND NOT "Modbus_Master_DB".BUSY,   // Modbus_Master
                          MB_ADDR := 1,
                          MODE := 0,
                          DATA_ADDR := 32067,
                          DATA_LEN := 1,
                          DATA_PTR := "Modbus_Send_Receive_1".Reading_Struct."32067",
                          DONE => "Modbus".Done,
                          BUSY => "Modbus".Busy,
                          ERROR => "Modbus".Error,
                          STATUS => "Modbus".Status);
   END_IF;
END_REGION

REGION Network 62: RD 32068
   RUNG wire#powerrail
      { S7_Templates := "SrcType := Int" } EQ_Contact(in1 := "IEC_Counter_0_DB".CV, in2 := 57)
      { S7_Templates := "[card := 0, word_type := UInt, dword_type := UDInt, byte_type := USInt, any_type := Variant]" } "Modbus_Master_DB".Modbus_Master(REQ := wire#w1, MB_ADDR := 1, MODE := 0, DATA_ADDR := 32068, DATA_LEN := 1, DATA_PTR := "Modbus_Send_Receive_1".Reading_Struct."32068", DONE => "Modbus".Done, BUSY => "Modbus".Busy, ERROR => "Modbus".Error, STATUS => "Modbus".Status)
   END_RUNG
   RUNG wire#powerrail
      Contact( "Comm_ok" )
      { S7_Templates := "SrcType := Int" } EQ_Contact(in1 := "IEC_Counter_0_DB".CV, in2 := 57)
      I_Contact( "Modbus_Master_DB".BUSY )
   END_RUNG wire#w1
   // the same network as SCL:
   IF "IEC_Counter_0_DB".CV = 57 THEN
       "Modbus_Master_DB"(REQ := "Comm_ok" AND ("IEC_Counter_0_DB".CV = 57) AND NOT "Modbus_Master_DB".BUSY,   // Modbus_Master
                          MB_ADDR := 1,
                          MODE := 0,
                          DATA_ADDR := 32068,
                          DATA_LEN := 1,
                          DATA_PTR := "Modbus_Send_Receive_1".Reading_Struct."32068",
                          DONE => "Modbus".Done,
                          BUSY => "Modbus".Busy,
                          ERROR => "Modbus".Error,
                          STATUS => "Modbus".Status);
   END_IF;
END_REGION

REGION Network 63: RD 32069
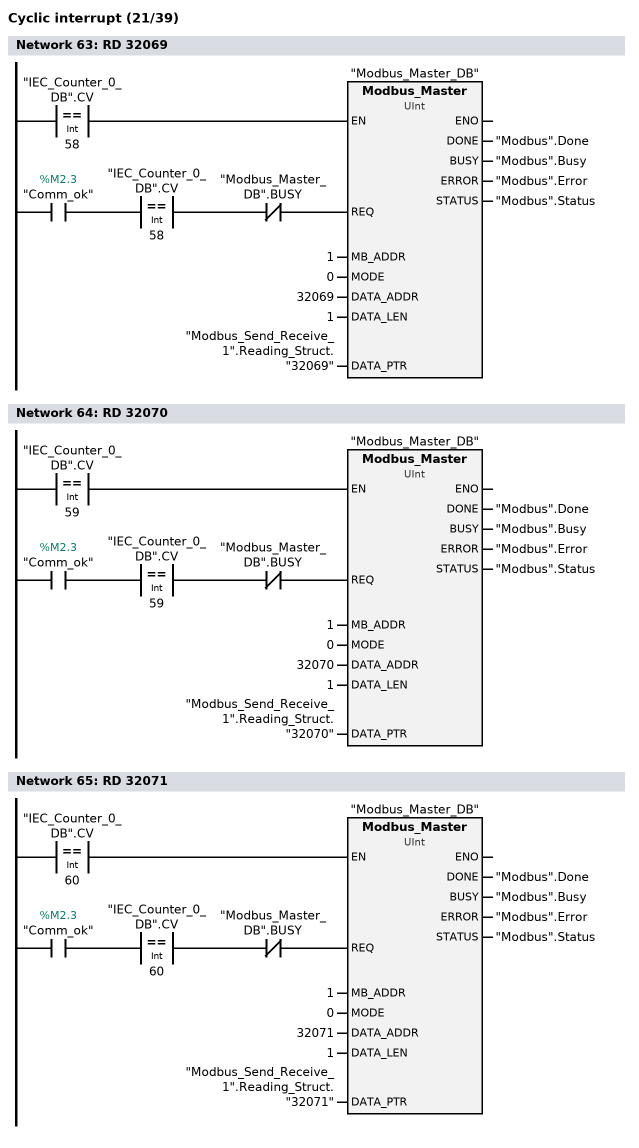
   RUNG wire#powerrail
      { S7_Templates := "SrcType := Int" } EQ_Contact(in1 := "IEC_Counter_0_DB".CV, in2 := 58)
      { S7_Templates := "[card := 0, word_type := UInt, dword_type := UDInt, byte_type := USInt, any_type := Variant]" } "Modbus_Master_DB".Modbus_Master(REQ := wire#w1, MB_ADDR := 1, MODE := 0, DATA_ADDR := 32069, DATA_LEN := 1, DATA_PTR := "Modbus_Send_Receive_1".Reading_Struct."32069", DONE => "Modbus".Done, BUSY => "Modbus".Busy, ERROR => "Modbus".Error, STATUS => "Modbus".Status)
   END_RUNG
   RUNG wire#powerrail
      Contact( "Comm_ok" )
      { S7_Templates := "SrcType := Int" } EQ_Contact(in1 := "IEC_Counter_0_DB".CV, in2 := 58)
      I_Contact( "Modbus_Master_DB".BUSY )
   END_RUNG wire#w1
   // the same network as SCL:
   IF "IEC_Counter_0_DB".CV = 58 THEN
       "Modbus_Master_DB"(REQ := "Comm_ok" AND ("IEC_Counter_0_DB".CV = 58) AND NOT "Modbus_Master_DB".BUSY,   // Modbus_Master
                          MB_ADDR := 1,
                          MODE := 0,
                          DATA_ADDR := 32069,
                          DATA_LEN := 1,
                          DATA_PTR := "Modbus_Send_Receive_1".Reading_Struct."32069",
                          DONE => "Modbus".Done,
                          BUSY => "Modbus".Busy,
                          ERROR => "Modbus".Error,
                          STATUS => "Modbus".Status);
   END_IF;
END_REGION

REGION Network 64: RD 32070
   RUNG wire#powerrail
      { S7_Templates := "SrcType := Int" } EQ_Contact(in1 := "IEC_Counter_0_DB".CV, in2 := 59)
      { S7_Templates := "[card := 0, word_type := UInt, dword_type := UDInt, byte_type := USInt, any_type := Variant]" } "Modbus_Master_DB".Modbus_Master(REQ := wire#w1, MB_ADDR := 1, MODE := 0, DATA_ADDR := 32070, DATA_LEN := 1, DATA_PTR := "Modbus_Send_Receive_1".Reading_Struct."32070", DONE => "Modbus".Done, BUSY => "Modbus".Busy, ERROR => "Modbus".Error, STATUS => "Modbus".Status)
   END_RUNG
   RUNG wire#powerrail
      Contact( "Comm_ok" )
      { S7_Templates := "SrcType := Int" } EQ_Contact(in1 := "IEC_Counter_0_DB".CV, in2 := 59)
      I_Contact( "Modbus_Master_DB".BUSY )
   END_RUNG wire#w1
   // the same network as SCL:
   IF "IEC_Counter_0_DB".CV = 59 THEN
       "Modbus_Master_DB"(REQ := "Comm_ok" AND ("IEC_Counter_0_DB".CV = 59) AND NOT "Modbus_Master_DB".BUSY,   // Modbus_Master
                          MB_ADDR := 1,
                          MODE := 0,
                          DATA_ADDR := 32070,
                          DATA_LEN := 1,
                          DATA_PTR := "Modbus_Send_Receive_1".Reading_Struct."32070",
                          DONE => "Modbus".Done,
                          BUSY => "Modbus".Busy,
                          ERROR => "Modbus".Error,
                          STATUS => "Modbus".Status);
   END_IF;
END_REGION

REGION Network 65: RD 32071
   RUNG wire#powerrail
      { S7_Templates := "SrcType := Int" } EQ_Contact(in1 := "IEC_Counter_0_DB".CV, in2 := 60)
      { S7_Templates := "[card := 0, word_type := UInt, dword_type := UDInt, byte_type := USInt, any_type := Variant]" } "Modbus_Master_DB".Modbus_Master(REQ := wire#w1, MB_ADDR := 1, MODE := 0, DATA_ADDR := 32071, DATA_LEN := 1, DATA_PTR := "Modbus_Send_Receive_1".Reading_Struct."32071", DONE => "Modbus".Done, BUSY => "Modbus".Busy, ERROR => "Modbus".Error, STATUS => "Modbus".Status)
   END_RUNG
   RUNG wire#powerrail
      Contact( "Comm_ok" )
      { S7_Templates := "SrcType := Int" } EQ_Contact(in1 := "IEC_Counter_0_DB".CV, in2 := 60)
      I_Contact( "Modbus_Master_DB".BUSY )
   END_RUNG wire#w1
   // the same network as SCL:
   IF "IEC_Counter_0_DB".CV = 60 THEN
       "Modbus_Master_DB"(REQ := "Comm_ok" AND ("IEC_Counter_0_DB".CV = 60) AND NOT "Modbus_Master_DB".BUSY,   // Modbus_Master
                          MB_ADDR := 1,
                          MODE := 0,
                          DATA_ADDR := 32071,
                          DATA_LEN := 1,
                          DATA_PTR := "Modbus_Send_Receive_1".Reading_Struct."32071",
                          DONE => "Modbus".Done,
                          BUSY => "Modbus".Busy,
                          ERROR => "Modbus".Error,
                          STATUS => "Modbus".Status);
   END_IF;
END_REGION

REGION Network 66: RD 32073
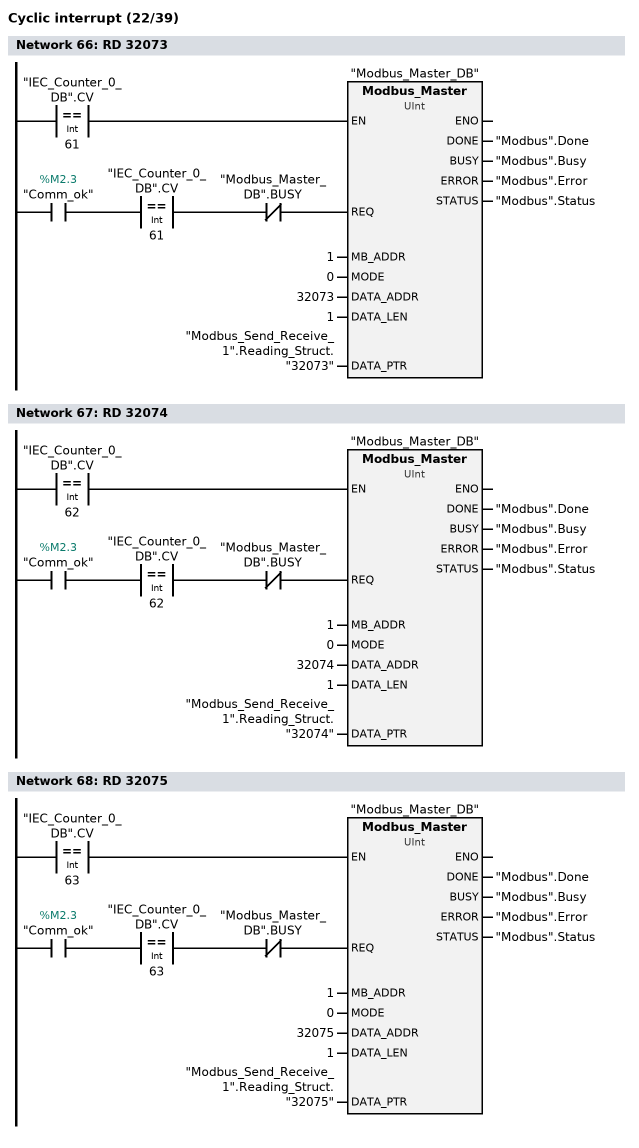
   RUNG wire#powerrail
      { S7_Templates := "SrcType := Int" } EQ_Contact(in1 := "IEC_Counter_0_DB".CV, in2 := 61)
      { S7_Templates := "[card := 0, word_type := UInt, dword_type := UDInt, byte_type := USInt, any_type := Variant]" } "Modbus_Master_DB".Modbus_Master(REQ := wire#w1, MB_ADDR := 1, MODE := 0, DATA_ADDR := 32073, DATA_LEN := 1, DATA_PTR := "Modbus_Send_Receive_1".Reading_Struct."32073", DONE => "Modbus".Done, BUSY => "Modbus".Busy, ERROR => "Modbus".Error, STATUS => "Modbus".Status)
   END_RUNG
   RUNG wire#powerrail
      Contact( "Comm_ok" )
      { S7_Templates := "SrcType := Int" } EQ_Contact(in1 := "IEC_Counter_0_DB".CV, in2 := 61)
      I_Contact( "Modbus_Master_DB".BUSY )
   END_RUNG wire#w1
   // the same network as SCL:
   IF "IEC_Counter_0_DB".CV = 61 THEN
       "Modbus_Master_DB"(REQ := "Comm_ok" AND ("IEC_Counter_0_DB".CV = 61) AND NOT "Modbus_Master_DB".BUSY,   // Modbus_Master
                          MB_ADDR := 1,
                          MODE := 0,
                          DATA_ADDR := 32073,
                          DATA_LEN := 1,
                          DATA_PTR := "Modbus_Send_Receive_1".Reading_Struct."32073",
                          DONE => "Modbus".Done,
                          BUSY => "Modbus".Busy,
                          ERROR => "Modbus".Error,
                          STATUS => "Modbus".Status);
   END_IF;
END_REGION

REGION Network 67: RD 32074
   RUNG wire#powerrail
      { S7_Templates := "SrcType := Int" } EQ_Contact(in1 := "IEC_Counter_0_DB".CV, in2 := 62)
      { S7_Templates := "[card := 0, word_type := UInt, dword_type := UDInt, byte_type := USInt, any_type := Variant]" } "Modbus_Master_DB".Modbus_Master(REQ := wire#w1, MB_ADDR := 1, MODE := 0, DATA_ADDR := 32074, DATA_LEN := 1, DATA_PTR := "Modbus_Send_Receive_1".Reading_Struct."32074", DONE => "Modbus".Done, BUSY => "Modbus".Busy, ERROR => "Modbus".Error, STATUS => "Modbus".Status)
   END_RUNG
   RUNG wire#powerrail
      Contact( "Comm_ok" )
      { S7_Templates := "SrcType := Int" } EQ_Contact(in1 := "IEC_Counter_0_DB".CV, in2 := 62)
      I_Contact( "Modbus_Master_DB".BUSY )
   END_RUNG wire#w1
   // the same network as SCL:
   IF "IEC_Counter_0_DB".CV = 62 THEN
       "Modbus_Master_DB"(REQ := "Comm_ok" AND ("IEC_Counter_0_DB".CV = 62) AND NOT "Modbus_Master_DB".BUSY,   // Modbus_Master
                          MB_ADDR := 1,
                          MODE := 0,
                          DATA_ADDR := 32074,
                          DATA_LEN := 1,
                          DATA_PTR := "Modbus_Send_Receive_1".Reading_Struct."32074",
                          DONE => "Modbus".Done,
                          BUSY => "Modbus".Busy,
                          ERROR => "Modbus".Error,
                          STATUS => "Modbus".Status);
   END_IF;
END_REGION

REGION Network 68: RD 32075
   RUNG wire#powerrail
      { S7_Templates := "SrcType := Int" } EQ_Contact(in1 := "IEC_Counter_0_DB".CV, in2 := 63)
      { S7_Templates := "[card := 0, word_type := UInt, dword_type := UDInt, byte_type := USInt, any_type := Variant]" } "Modbus_Master_DB".Modbus_Master(REQ := wire#w1, MB_ADDR := 1, MODE := 0, DATA_ADDR := 32075, DATA_LEN := 1, DATA_PTR := "Modbus_Send_Receive_1".Reading_Struct."32075", DONE => "Modbus".Done, BUSY => "Modbus".Busy, ERROR => "Modbus".Error, STATUS => "Modbus".Status)
   END_RUNG
   RUNG wire#powerrail
      Contact( "Comm_ok" )
      { S7_Templates := "SrcType := Int" } EQ_Contact(in1 := "IEC_Counter_0_DB".CV, in2 := 63)
      I_Contact( "Modbus_Master_DB".BUSY )
   END_RUNG wire#w1
   // the same network as SCL:
   IF "IEC_Counter_0_DB".CV = 63 THEN
       "Modbus_Master_DB"(REQ := "Comm_ok" AND ("IEC_Counter_0_DB".CV = 63) AND NOT "Modbus_Master_DB".BUSY,   // Modbus_Master
                          MB_ADDR := 1,
                          MODE := 0,
                          DATA_ADDR := 32075,
                          DATA_LEN := 1,
                          DATA_PTR := "Modbus_Send_Receive_1".Reading_Struct."32075",
                          DONE => "Modbus".Done,
                          BUSY => "Modbus".Busy,
                          ERROR => "Modbus".Error,
                          STATUS => "Modbus".Status);
   END_IF;
END_REGION

REGION Network 69: RD 32076
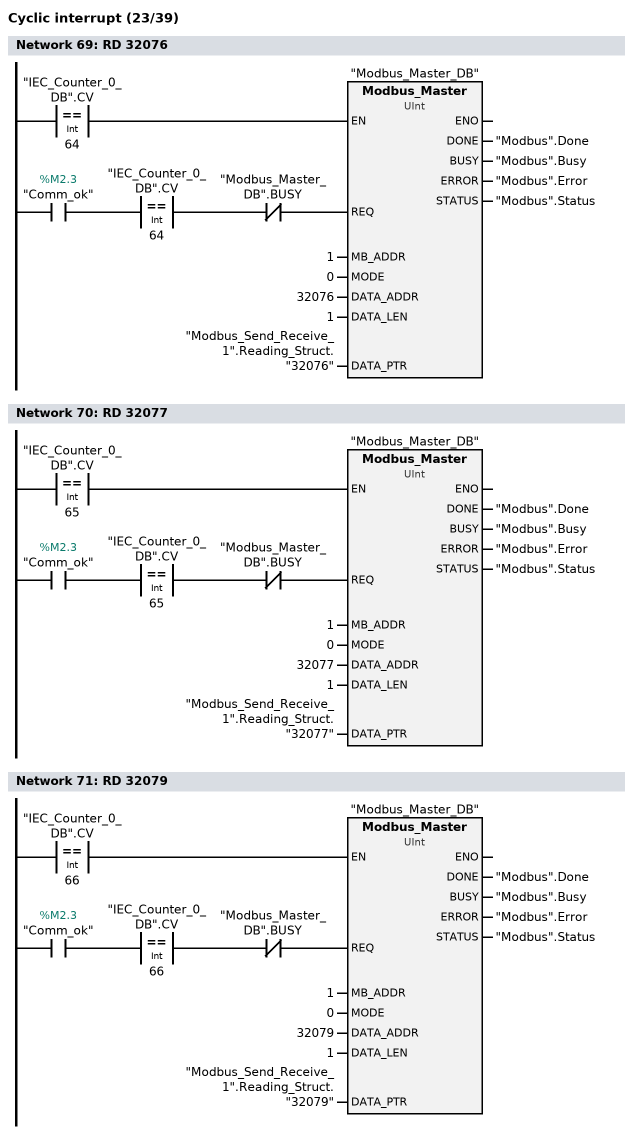
   RUNG wire#powerrail
      { S7_Templates := "SrcType := Int" } EQ_Contact(in1 := "IEC_Counter_0_DB".CV, in2 := 64)
      { S7_Templates := "[card := 0, word_type := UInt, dword_type := UDInt, byte_type := USInt, any_type := Variant]" } "Modbus_Master_DB".Modbus_Master(REQ := wire#w1, MB_ADDR := 1, MODE := 0, DATA_ADDR := 32076, DATA_LEN := 1, DATA_PTR := "Modbus_Send_Receive_1".Reading_Struct."32076", DONE => "Modbus".Done, BUSY => "Modbus".Busy, ERROR => "Modbus".Error, STATUS => "Modbus".Status)
   END_RUNG
   RUNG wire#powerrail
      Contact( "Comm_ok" )
      { S7_Templates := "SrcType := Int" } EQ_Contact(in1 := "IEC_Counter_0_DB".CV, in2 := 64)
      I_Contact( "Modbus_Master_DB".BUSY )
   END_RUNG wire#w1
   // the same network as SCL:
   IF "IEC_Counter_0_DB".CV = 64 THEN
       "Modbus_Master_DB"(REQ := "Comm_ok" AND ("IEC_Counter_0_DB".CV = 64) AND NOT "Modbus_Master_DB".BUSY,   // Modbus_Master
                          MB_ADDR := 1,
                          MODE := 0,
                          DATA_ADDR := 32076,
                          DATA_LEN := 1,
                          DATA_PTR := "Modbus_Send_Receive_1".Reading_Struct."32076",
                          DONE => "Modbus".Done,
                          BUSY => "Modbus".Busy,
                          ERROR => "Modbus".Error,
                          STATUS => "Modbus".Status);
   END_IF;
END_REGION

REGION Network 70: RD 32077
   RUNG wire#powerrail
      { S7_Templates := "SrcType := Int" } EQ_Contact(in1 := "IEC_Counter_0_DB".CV, in2 := 65)
      { S7_Templates := "[card := 0, word_type := UInt, dword_type := UDInt, byte_type := USInt, any_type := Variant]" } "Modbus_Master_DB".Modbus_Master(REQ := wire#w1, MB_ADDR := 1, MODE := 0, DATA_ADDR := 32077, DATA_LEN := 1, DATA_PTR := "Modbus_Send_Receive_1".Reading_Struct."32077", DONE => "Modbus".Done, BUSY => "Modbus".Busy, ERROR => "Modbus".Error, STATUS => "Modbus".Status)
   END_RUNG
   RUNG wire#powerrail
      Contact( "Comm_ok" )
      { S7_Templates := "SrcType := Int" } EQ_Contact(in1 := "IEC_Counter_0_DB".CV, in2 := 65)
      I_Contact( "Modbus_Master_DB".BUSY )
   END_RUNG wire#w1
   // the same network as SCL:
   IF "IEC_Counter_0_DB".CV = 65 THEN
       "Modbus_Master_DB"(REQ := "Comm_ok" AND ("IEC_Counter_0_DB".CV = 65) AND NOT "Modbus_Master_DB".BUSY,   // Modbus_Master
                          MB_ADDR := 1,
                          MODE := 0,
                          DATA_ADDR := 32077,
                          DATA_LEN := 1,
                          DATA_PTR := "Modbus_Send_Receive_1".Reading_Struct."32077",
                          DONE => "Modbus".Done,
                          BUSY => "Modbus".Busy,
                          ERROR => "Modbus".Error,
                          STATUS => "Modbus".Status);
   END_IF;
END_REGION

REGION Network 71: RD 32079
   RUNG wire#powerrail
      { S7_Templates := "SrcType := Int" } EQ_Contact(in1 := "IEC_Counter_0_DB".CV, in2 := 66)
      { S7_Templates := "[card := 0, word_type := UInt, dword_type := UDInt, byte_type := USInt, any_type := Variant]" } "Modbus_Master_DB".Modbus_Master(REQ := wire#w1, MB_ADDR := 1, MODE := 0, DATA_ADDR := 32079, DATA_LEN := 1, DATA_PTR := "Modbus_Send_Receive_1".Reading_Struct."32079", DONE => "Modbus".Done, BUSY => "Modbus".Busy, ERROR => "Modbus".Error, STATUS => "Modbus".Status)
   END_RUNG
   RUNG wire#powerrail
      Contact( "Comm_ok" )
      { S7_Templates := "SrcType := Int" } EQ_Contact(in1 := "IEC_Counter_0_DB".CV, in2 := 66)
      I_Contact( "Modbus_Master_DB".BUSY )
   END_RUNG wire#w1
   // the same network as SCL:
   IF "IEC_Counter_0_DB".CV = 66 THEN
       "Modbus_Master_DB"(REQ := "Comm_ok" AND ("IEC_Counter_0_DB".CV = 66) AND NOT "Modbus_Master_DB".BUSY,   // Modbus_Master
                          MB_ADDR := 1,
                          MODE := 0,
                          DATA_ADDR := 32079,
                          DATA_LEN := 1,
                          DATA_PTR := "Modbus_Send_Receive_1".Reading_Struct."32079",
                          DONE => "Modbus".Done,
                          BUSY => "Modbus".Busy,
                          ERROR => "Modbus".Error,
                          STATUS => "Modbus".Status);
   END_IF;
END_REGION

REGION Network 72: RD 32080
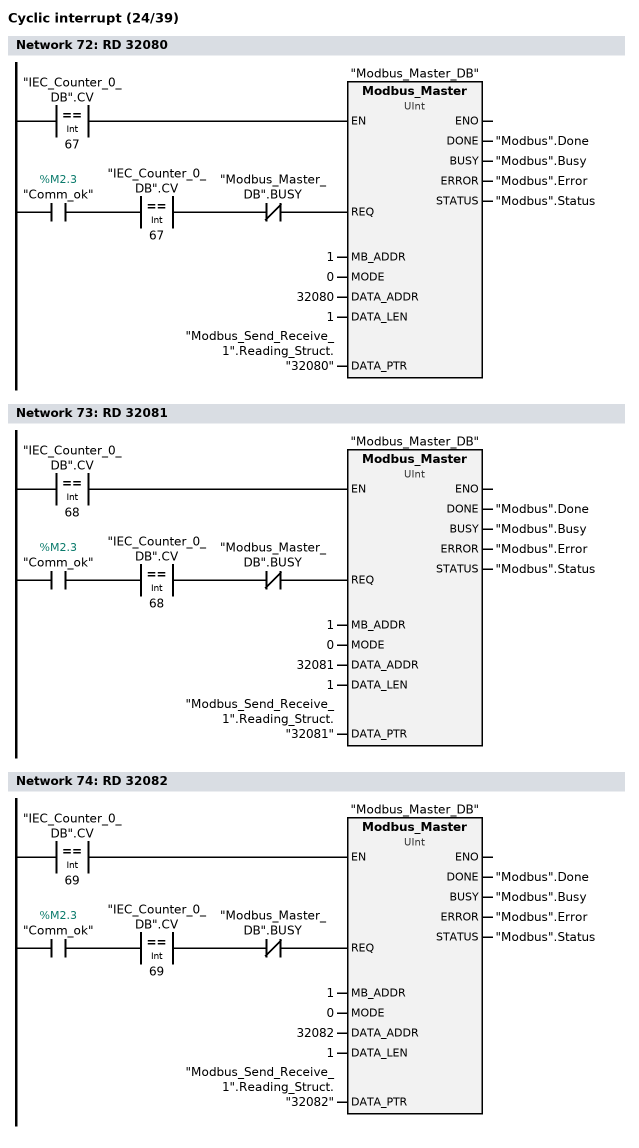
   RUNG wire#powerrail
      { S7_Templates := "SrcType := Int" } EQ_Contact(in1 := "IEC_Counter_0_DB".CV, in2 := 67)
      { S7_Templates := "[card := 0, word_type := UInt, dword_type := UDInt, byte_type := USInt, any_type := Variant]" } "Modbus_Master_DB".Modbus_Master(REQ := wire#w1, MB_ADDR := 1, MODE := 0, DATA_ADDR := 32080, DATA_LEN := 1, DATA_PTR := "Modbus_Send_Receive_1".Reading_Struct."32080", DONE => "Modbus".Done, BUSY => "Modbus".Busy, ERROR => "Modbus".Error, STATUS => "Modbus".Status)
   END_RUNG
   RUNG wire#powerrail
      Contact( "Comm_ok" )
      { S7_Templates := "SrcType := Int" } EQ_Contact(in1 := "IEC_Counter_0_DB".CV, in2 := 67)
      I_Contact( "Modbus_Master_DB".BUSY )
   END_RUNG wire#w1
   // the same network as SCL:
   IF "IEC_Counter_0_DB".CV = 67 THEN
       "Modbus_Master_DB"(REQ := "Comm_ok" AND ("IEC_Counter_0_DB".CV = 67) AND NOT "Modbus_Master_DB".BUSY,   // Modbus_Master
                          MB_ADDR := 1,
                          MODE := 0,
                          DATA_ADDR := 32080,
                          DATA_LEN := 1,
                          DATA_PTR := "Modbus_Send_Receive_1".Reading_Struct."32080",
                          DONE => "Modbus".Done,
                          BUSY => "Modbus".Busy,
                          ERROR => "Modbus".Error,
                          STATUS => "Modbus".Status);
   END_IF;
END_REGION

REGION Network 73: RD 32081
   RUNG wire#powerrail
      { S7_Templates := "SrcType := Int" } EQ_Contact(in1 := "IEC_Counter_0_DB".CV, in2 := 68)
      { S7_Templates := "[card := 0, word_type := UInt, dword_type := UDInt, byte_type := USInt, any_type := Variant]" } "Modbus_Master_DB".Modbus_Master(REQ := wire#w1, MB_ADDR := 1, MODE := 0, DATA_ADDR := 32081, DATA_LEN := 1, DATA_PTR := "Modbus_Send_Receive_1".Reading_Struct."32081", DONE => "Modbus".Done, BUSY => "Modbus".Busy, ERROR => "Modbus".Error, STATUS => "Modbus".Status)
   END_RUNG
   RUNG wire#powerrail
      Contact( "Comm_ok" )
      { S7_Templates := "SrcType := Int" } EQ_Contact(in1 := "IEC_Counter_0_DB".CV, in2 := 68)
      I_Contact( "Modbus_Master_DB".BUSY )
   END_RUNG wire#w1
   // the same network as SCL:
   IF "IEC_Counter_0_DB".CV = 68 THEN
       "Modbus_Master_DB"(REQ := "Comm_ok" AND ("IEC_Counter_0_DB".CV = 68) AND NOT "Modbus_Master_DB".BUSY,   // Modbus_Master
                          MB_ADDR := 1,
                          MODE := 0,
                          DATA_ADDR := 32081,
                          DATA_LEN := 1,
                          DATA_PTR := "Modbus_Send_Receive_1".Reading_Struct."32081",
                          DONE => "Modbus".Done,
                          BUSY => "Modbus".Busy,
                          ERROR => "Modbus".Error,
                          STATUS => "Modbus".Status);
   END_IF;
END_REGION

REGION Network 74: RD 32082
   RUNG wire#powerrail
      { S7_Templates := "SrcType := Int" } EQ_Contact(in1 := "IEC_Counter_0_DB".CV, in2 := 69)
      { S7_Templates := "[card := 0, word_type := UInt, dword_type := UDInt, byte_type := USInt, any_type := Variant]" } "Modbus_Master_DB".Modbus_Master(REQ := wire#w1, MB_ADDR := 1, MODE := 0, DATA_ADDR := 32082, DATA_LEN := 1, DATA_PTR := "Modbus_Send_Receive_1".Reading_Struct."32082", DONE => "Modbus".Done, BUSY => "Modbus".Busy, ERROR => "Modbus".Error, STATUS => "Modbus".Status)
   END_RUNG
   RUNG wire#powerrail
      Contact( "Comm_ok" )
      { S7_Templates := "SrcType := Int" } EQ_Contact(in1 := "IEC_Counter_0_DB".CV, in2 := 69)
      I_Contact( "Modbus_Master_DB".BUSY )
   END_RUNG wire#w1
   // the same network as SCL:
   IF "IEC_Counter_0_DB".CV = 69 THEN
       "Modbus_Master_DB"(REQ := "Comm_ok" AND ("IEC_Counter_0_DB".CV = 69) AND NOT "Modbus_Master_DB".BUSY,   // Modbus_Master
                          MB_ADDR := 1,
                          MODE := 0,
                          DATA_ADDR := 32082,
                          DATA_LEN := 1,
                          DATA_PTR := "Modbus_Send_Receive_1".Reading_Struct."32082",
                          DONE => "Modbus".Done,
                          BUSY => "Modbus".Busy,
                          ERROR => "Modbus".Error,
                          STATUS => "Modbus".Status);
   END_IF;
END_REGION

REGION Network 75: RD 32083
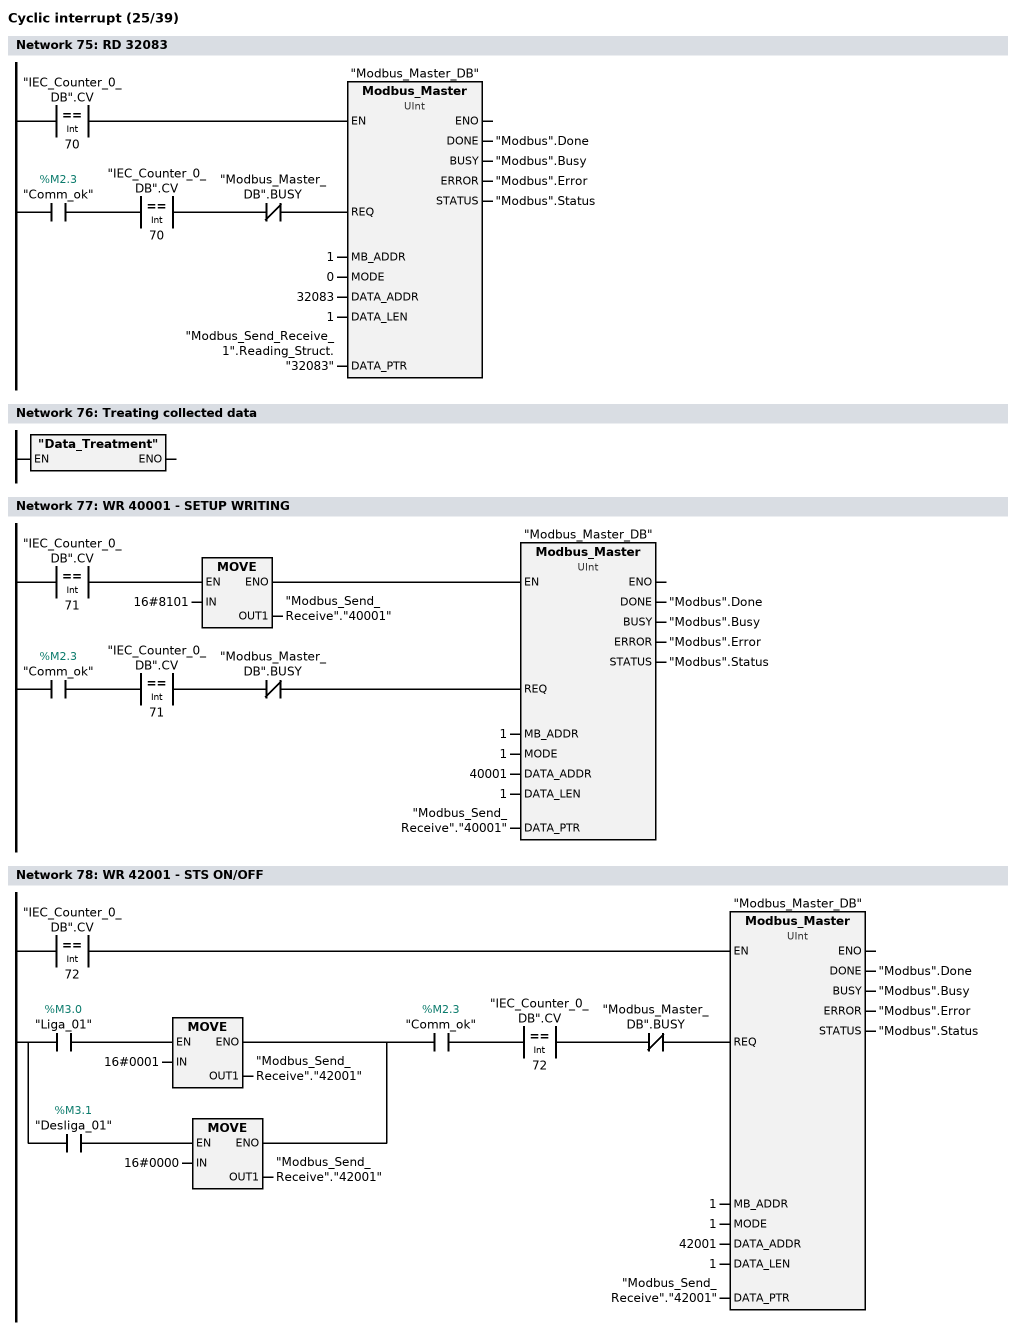
   RUNG wire#powerrail
      { S7_Templates := "SrcType := Int" } EQ_Contact(in1 := "IEC_Counter_0_DB".CV, in2 := 70)
      { S7_Templates := "[card := 0, word_type := UInt, dword_type := UDInt, byte_type := USInt, any_type := Variant]" } "Modbus_Master_DB".Modbus_Master(REQ := wire#w1, MB_ADDR := 1, MODE := 0, DATA_ADDR := 32083, DATA_LEN := 1, DATA_PTR := "Modbus_Send_Receive_1".Reading_Struct."32083", DONE => "Modbus".Done, BUSY => "Modbus".Busy, ERROR => "Modbus".Error, STATUS => "Modbus".Status)
   END_RUNG
   RUNG wire#powerrail
      Contact( "Comm_ok" )
      { S7_Templates := "SrcType := Int" } EQ_Contact(in1 := "IEC_Counter_0_DB".CV, in2 := 70)
      I_Contact( "Modbus_Master_DB".BUSY )
   END_RUNG wire#w1
   // the same network as SCL:
   IF "IEC_Counter_0_DB".CV = 70 THEN
       "Modbus_Master_DB"(REQ := "Comm_ok" AND ("IEC_Counter_0_DB".CV = 70) AND NOT "Modbus_Master_DB".BUSY,   // Modbus_Master
                          MB_ADDR := 1,
                          MODE := 0,
                          DATA_ADDR := 32083,
                          DATA_LEN := 1,
                          DATA_PTR := "Modbus_Send_Receive_1".Reading_Struct."32083",
                          DONE => "Modbus".Done,
                          BUSY => "Modbus".Busy,
                          ERROR => "Modbus".Error,
                          STATUS => "Modbus".Status);
   END_IF;
END_REGION

REGION Network 76: Treating collected data
   RUNG wire#powerrail
      "Data_Treatment"()
   END_RUNG
   // the same network as SCL:
   "Data_Treatment"();
END_REGION

